   STATUS[774].EXT.BIT19 := FALSE;
   STATUS[774].EXT.BIT20 := FALSE;
   STATUS[774].EXT.AlarmSuppressed := FALSE;
   STATUS[774].EXT.AlarmPrsent := FALSE;
   STATUS[774].EXT.AlarmFailUnAck := FALSE;
   STATUS[774].Status := 0;
   STATUS[774].TimeStamp := 16#0000;
   STATUS[775].VALUE := 0.0;
   STATUS[775].TRIGVALUE := 0.0;
   STATUS[775].EXT.AlarmWarnUnAck := FALSE;
   STATUS[775].EXT.AckRequired := FALSE;
   STATUS[775].EXT.Maintanence := FALSE;
   STATUS[775].EXT.Operation := FALSE;
   STATUS[775].EXT.Forced := FALSE;
   STATUS[775].EXT.BIT29 := FALSE;
   STATUS[775].EXT.BIT30 := FALSE;
   STATUS[775].EXT.BIT31 := FALSE;
   STATUS[775].EXT.ModeBit1 := FALSE;
   STATUS[775].EXT.ModeBit2 := FALSE;
   STATUS[775].EXT.ModeBit3 := FALSE;
   STATUS[775].EXT.BIT19 := FALSE;
   STATUS[775].EXT.BIT20 := FALSE;
   STATUS[775].EXT.AlarmSuppressed := FALSE;
   STATUS[775].EXT.AlarmPrsent := FALSE;
   STATUS[775].EXT.AlarmFailUnAck := FALSE;
   STATUS[775].Status := 0;
   STATUS[775].TimeStamp := 16#0000;
   STATUS[776].VALUE := 0.0;
   STATUS[776].TRIGVALUE := 0.0;
   STATUS[776].EXT.AlarmWarnUnAck := FALSE;
   STATUS[776].EXT.AckRequired := FALSE;
   STATUS[776].EXT.Maintanence := FALSE;
   STATUS[776].EXT.Operation := FALSE;
   STATUS[776].EXT.Forced := FALSE;
   STATUS[776].EXT.BIT29 := FALSE;
   STATUS[776].EXT.BIT30 := FALSE;
   STATUS[776].EXT.BIT31 := FALSE;
   STATUS[776].EXT.ModeBit1 := FALSE;
   STATUS[776].EXT.ModeBit2 := FALSE;
   STATUS[776].EXT.ModeBit3 := FALSE;
   STATUS[776].EXT.BIT19 := FALSE;
   STATUS[776].EXT.BIT20 := FALSE;
   STATUS[776].EXT.AlarmSuppressed := FALSE;
   STATUS[776].EXT.AlarmPrsent := FALSE;
   STATUS[776].EXT.AlarmFailUnAck := FALSE;
   STATUS[776].Status := 0;
   STATUS[776].TimeStamp := 16#0000;
   STATUS[777].VALUE := 0.0;
   STATUS[777].TRIGVALUE := 0.0;
   STATUS[777].EXT.AlarmWarnUnAck := FALSE;
   STATUS[777].EXT.AckRequired := FALSE;
   STATUS[777].EXT.Maintanence := FALSE;
   STATUS[777].EXT.Operation := FALSE;
   STATUS[777].EXT.Forced := FALSE;
   STATUS[777].EXT.BIT29 := FALSE;
   STATUS[777].EXT.BIT30 := FALSE;
   STATUS[777].EXT.BIT31 := FALSE;
   STATUS[777].EXT.ModeBit1 := FALSE;
   STATUS[777].EXT.ModeBit2 := FALSE;
   STATUS[777].EXT.ModeBit3 := FALSE;
   STATUS[777].EXT.BIT19 := FALSE;
   STATUS[777].EXT.BIT20 := FALSE;
   STATUS[777].EXT.AlarmSuppressed := FALSE;
   STATUS[777].EXT.AlarmPrsent := FALSE;
   STATUS[777].EXT.AlarmFailUnAck := FALSE;
   STATUS[777].Status := 0;
   STATUS[777].TimeStamp := 16#0000;
   STATUS[778].VALUE := 0.0;
   STATUS[778].TRIGVALUE := 0.0;
   STATUS[778].EXT.AlarmWarnUnAck := FALSE;
   STATUS[778].EXT.AckRequired := FALSE;
   STATUS[778].EXT.Maintanence := FALSE;
   STATUS[778].EXT.Operation := FALSE;
   STATUS[778].EXT.Forced := FALSE;
   STATUS[778].EXT.BIT29 := FALSE;
   STATUS[778].EXT.BIT30 := FALSE;
   STATUS[778].EXT.BIT31 := FALSE;
   STATUS[778].EXT.ModeBit1 := FALSE;
   STATUS[778].EXT.ModeBit2 := FALSE;
   STATUS[778].EXT.ModeBit3 := FALSE;
   STATUS[778].EXT.BIT19 := FALSE;
   STATUS[778].EXT.BIT20 := FALSE;
   STATUS[778].EXT.AlarmSuppressed := FALSE;
   STATUS[778].EXT.AlarmPrsent := FALSE;
   STATUS[778].EXT.AlarmFailUnAck := FALSE;
   STATUS[778].Status := 0;
   STATUS[778].TimeStamp := 16#0000;
   STATUS[779].VALUE := 0.0;
   STATUS[779].TRIGVALUE := 0.0;
   STATUS[779].EXT.AlarmWarnUnAck := FALSE;
   STATUS[779].EXT.AckRequired := FALSE;
   STATUS[779].EXT.Maintanence := FALSE;
   STATUS[779].EXT.Operation := FALSE;
   STATUS[779].EXT.Forced := FALSE;
   STATUS[779].EXT.BIT29 := FALSE;
   STATUS[779].EXT.BIT30 := FALSE;
   STATUS[779].EXT.BIT31 := FALSE;
   STATUS[779].EXT.ModeBit1 := FALSE;
   STATUS[779].EXT.ModeBit2 := FALSE;
   STATUS[779].EXT.ModeBit3 := FALSE;
   STATUS[779].EXT.BIT19 := FALSE;
   STATUS[779].EXT.BIT20 := FALSE;
   STATUS[779].EXT.AlarmSuppressed := FALSE;
   STATUS[779].EXT.AlarmPrsent := FALSE;
   STATUS[779].EXT.AlarmFailUnAck := FALSE;
   STATUS[779].Status := 0;
   STATUS[779].TimeStamp := 16#0000;
   STATUS[780].VALUE := 0.0;
   STATUS[780].TRIGVALUE := 0.0;
   STATUS[780].EXT.AlarmWarnUnAck := FALSE;
   STATUS[780].EXT.AckRequired := FALSE;
   STATUS[780].EXT.Maintanence := FALSE;
   STATUS[780].EXT.Operation := FALSE;
   STATUS[780].EXT.Forced := FALSE;
   STATUS[780].EXT.BIT29 := FALSE;
   STATUS[780].EXT.BIT30 := FALSE;
   STATUS[780].EXT.BIT31 := FALSE;
   STATUS[780].EXT.ModeBit1 := FALSE;
   STATUS[780].EXT.ModeBit2 := FALSE;
   STATUS[780].EXT.ModeBit3 := FALSE;
   STATUS[780].EXT.BIT19 := FALSE;
   STATUS[780].EXT.BIT20 := FALSE;
   STATUS[780].EXT.AlarmSuppressed := FALSE;
   STATUS[780].EXT.AlarmPrsent := FALSE;
   STATUS[780].EXT.AlarmFailUnAck := FALSE;
   STATUS[780].Status := 0;
   STATUS[780].TimeStamp := 16#0000;
   STATUS[781].VALUE := 0.0;
   STATUS[781].TRIGVALUE := 0.0;
   STATUS[781].EXT.AlarmWarnUnAck := FALSE;
   STATUS[781].EXT.AckRequired := FALSE;
   STATUS[781].EXT.Maintanence := FALSE;
   STATUS[781].EXT.Operation := FALSE;
   STATUS[781].EXT.Forced := FALSE;
   STATUS[781].EXT.BIT29 := FALSE;
   STATUS[781].EXT.BIT30 := FALSE;
   STATUS[781].EXT.BIT31 := FALSE;
   STATUS[781].EXT.ModeBit1 := FALSE;
   STATUS[781].EXT.ModeBit2 := FALSE;
   STATUS[781].EXT.ModeBit3 := FALSE;
   STATUS[781].EXT.BIT19 := FALSE;
   STATUS[781].EXT.BIT20 := FALSE;
   STATUS[781].EXT.AlarmSuppressed := FALSE;
   STATUS[781].EXT.AlarmPrsent := FALSE;
   STATUS[781].EXT.AlarmFailUnAck := FALSE;
   STATUS[781].Status := 0;
   STATUS[781].TimeStamp := 16#0000;
   STATUS[782].VALUE := 0.0;
   STATUS[782].TRIGVALUE := 0.0;
   STATUS[782].EXT.AlarmWarnUnAck := FALSE;
   STATUS[782].EXT.AckRequired := FALSE;
   STATUS[782].EXT.Maintanence := FALSE;
   STATUS[782].EXT.Operation := FALSE;
   STATUS[782].EXT.Forced := FALSE;
   STATUS[782].EXT.BIT29 := FALSE;
   STATUS[782].EXT.BIT30 := FALSE;
   STATUS[782].EXT.BIT31 := FALSE;
   STATUS[782].EXT.ModeBit1 := FALSE;
   STATUS[782].EXT.ModeBit2 := FALSE;
   STATUS[782].EXT.ModeBit3 := FALSE;
   STATUS[782].EXT.BIT19 := FALSE;
   STATUS[782].EXT.BIT20 := FALSE;
   STATUS[782].EXT.AlarmSuppressed := FALSE;
   STATUS[782].EXT.AlarmPrsent := FALSE;
   STATUS[782].EXT.AlarmFailUnAck := FALSE;
   STATUS[782].Status := 0;
   STATUS[782].TimeStamp := 16#0000;
   STATUS[783].VALUE := 0.0;
   STATUS[783].TRIGVALUE := 0.0;
   STATUS[783].EXT.AlarmWarnUnAck := FALSE;
   STATUS[783].EXT.AckRequired := FALSE;
   STATUS[783].EXT.Maintanence := FALSE;
   STATUS[783].EXT.Operation := FALSE;
   STATUS[783].EXT.Forced := FALSE;
   STATUS[783].EXT.BIT29 := FALSE;
   STATUS[783].EXT.BIT30 := FALSE;
   STATUS[783].EXT.BIT31 := FALSE;
   STATUS[783].EXT.ModeBit1 := FALSE;
   STATUS[783].EXT.ModeBit2 := FALSE;
   STATUS[783].EXT.ModeBit3 := FALSE;
   STATUS[783].EXT.BIT19 := FALSE;
   STATUS[783].EXT.BIT20 := FALSE;
   STATUS[783].EXT.AlarmSuppressed := FALSE;
   STATUS[783].EXT.AlarmPrsent := FALSE;
   STATUS[783].EXT.AlarmFailUnAck := FALSE;
   STATUS[783].Status := 0;
   STATUS[783].TimeStamp := 16#0000;
   STATUS[784].VALUE := 0.0;
   STATUS[784].TRIGVALUE := 0.0;
   STATUS[784].EXT.AlarmWarnUnAck := FALSE;
   STATUS[784].EXT.AckRequired := FALSE;
   STATUS[784].EXT.Maintanence := FALSE;
   STATUS[784].EXT.Operation := FALSE;
   STATUS[784].EXT.Forced := FALSE;
   STATUS[784].EXT.BIT29 := FALSE;
   STATUS[784].EXT.BIT30 := FALSE;
   STATUS[784].EXT.BIT31 := FALSE;
   STATUS[784].EXT.ModeBit1 := FALSE;
   STATUS[784].EXT.ModeBit2 := FALSE;
   STATUS[784].EXT.ModeBit3 := FALSE;
   STATUS[784].EXT.BIT19 := FALSE;
   STATUS[784].EXT.BIT20 := FALSE;
   STATUS[784].EXT.AlarmSuppressed := FALSE;
   STATUS[784].EXT.AlarmPrsent := FALSE;
   STATUS[784].EXT.AlarmFailUnAck := FALSE;
   STATUS[784].Status := 0;
   STATUS[784].TimeStamp := 16#0000;
   STATUS[785].VALUE := 0.0;
   STATUS[785].TRIGVALUE := 0.0;
   STATUS[785].EXT.AlarmWarnUnAck := FALSE;
   STATUS[785].EXT.AckRequired := FALSE;
   STATUS[785].EXT.Maintanence := FALSE;
   STATUS[785].EXT.Operation := FALSE;
   STATUS[785].EXT.Forced := FALSE;
   STATUS[785].EXT.BIT29 := FALSE;
   STATUS[785].EXT.BIT30 := FALSE;
   STATUS[785].EXT.BIT31 := FALSE;
   STATUS[785].EXT.ModeBit1 := FALSE;
   STATUS[785].EXT.ModeBit2 := FALSE;
   STATUS[785].EXT.ModeBit3 := FALSE;
   STATUS[785].EXT.BIT19 := FALSE;
   STATUS[785].EXT.BIT20 := FALSE;
   STATUS[785].EXT.AlarmSuppressed := FALSE;
   STATUS[785].EXT.AlarmPrsent := FALSE;
   STATUS[785].EXT.AlarmFailUnAck := FALSE;
   STATUS[785].Status := 0;
   STATUS[785].TimeStamp := 16#0000;
   STATUS[786].VALUE := 0.0;
   STATUS[786].TRIGVALUE := 0.0;
   STATUS[786].EXT.AlarmWarnUnAck := FALSE;
   STATUS[786].EXT.AckRequired := FALSE;
   STATUS[786].EXT.Maintanence := FALSE;
   STATUS[786].EXT.Operation := FALSE;
   STATUS[786].EXT.Forced := FALSE;
   STATUS[786].EXT.BIT29 := FALSE;
   STATUS[786].EXT.BIT30 := FALSE;
   STATUS[786].EXT.BIT31 := FALSE;
   STATUS[786].EXT.ModeBit1 := FALSE;
   STATUS[786].EXT.ModeBit2 := FALSE;
   STATUS[786].EXT.ModeBit3 := FALSE;
   STATUS[786].EXT.BIT19 := FALSE;
   STATUS[786].EXT.BIT20 := FALSE;
   STATUS[786].EXT.AlarmSuppressed := FALSE;
   STATUS[786].EXT.AlarmPrsent := FALSE;
   STATUS[786].EXT.AlarmFailUnAck := FALSE;
   STATUS[786].Status := 0;
   STATUS[786].TimeStamp := 16#0000;
   STATUS[787].VALUE := 0.0;
   STATUS[787].TRIGVALUE := 0.0;
   STATUS[787].EXT.AlarmWarnUnAck := FALSE;
   STATUS[787].EXT.AckRequired := FALSE;
   STATUS[787].EXT.Maintanence := FALSE;
   STATUS[787].EXT.Operation := FALSE;
   STATUS[787].EXT.Forced := FALSE;
   STATUS[787].EXT.BIT29 := FALSE;
   STATUS[787].EXT.BIT30 := FALSE;
   STATUS[787].EXT.BIT31 := FALSE;
   STATUS[787].EXT.ModeBit1 := FALSE;
   STATUS[787].EXT.ModeBit2 := FALSE;
   STATUS[787].EXT.ModeBit3 := FALSE;
   STATUS[787].EXT.BIT19 := FALSE;
   STATUS[787].EXT.BIT20 := FALSE;
   STATUS[787].EXT.AlarmSuppressed := FALSE;
   STATUS[787].EXT.AlarmPrsent := FALSE;
   STATUS[787].EXT.AlarmFailUnAck := FALSE;
   STATUS[787].Status := 0;
   STATUS[787].TimeStamp := 16#0000;
   STATUS[788].VALUE := 0.0;
   STATUS[788].TRIGVALUE := 0.0;
   STATUS[788].EXT.AlarmWarnUnAck := FALSE;
   STATUS[788].EXT.AckRequired := FALSE;
   STATUS[788].EXT.Maintanence := FALSE;
   STATUS[788].EXT.Operation := FALSE;
   STATUS[788].EXT.Forced := FALSE;
   STATUS[788].EXT.BIT29 := FALSE;
   STATUS[788].EXT.BIT30 := FALSE;
   STATUS[788].EXT.BIT31 := FALSE;
   STATUS[788].EXT.ModeBit1 := FALSE;
   STATUS[788].EXT.ModeBit2 := FALSE;
   STATUS[788].EXT.ModeBit3 := FALSE;
   STATUS[788].EXT.BIT19 := FALSE;
   STATUS[788].EXT.BIT20 := FALSE;
   STATUS[788].EXT.AlarmSuppressed := FALSE;
   STATUS[788].EXT.AlarmPrsent := FALSE;
   STATUS[788].EXT.AlarmFailUnAck := FALSE;
   STATUS[788].Status := 0;
   STATUS[788].TimeStamp := 16#0000;
   STATUS[789].VALUE := 0.0;
   STATUS[789].TRIGVALUE := 0.0;
   STATUS[789].EXT.AlarmWarnUnAck := FALSE;
   STATUS[789].EXT.AckRequired := FALSE;
   STATUS[789].EXT.Maintanence := FALSE;
   STATUS[789].EXT.Operation := FALSE;
   STATUS[789].EXT.Forced := FALSE;
   STATUS[789].EXT.BIT29 := FALSE;
   STATUS[789].EXT.BIT30 := FALSE;
   STATUS[789].EXT.BIT31 := FALSE;
   STATUS[789].EXT.ModeBit1 := FALSE;
   STATUS[789].EXT.ModeBit2 := FALSE;
   STATUS[789].EXT.ModeBit3 := FALSE;
   STATUS[789].EXT.BIT19 := FALSE;
   STATUS[789].EXT.BIT20 := FALSE;
   STATUS[789].EXT.AlarmSuppressed := FALSE;
   STATUS[789].EXT.AlarmPrsent := FALSE;
   STATUS[789].EXT.AlarmFailUnAck := FALSE;
   STATUS[789].Status := 0;
   STATUS[789].TimeStamp := 16#0000;
   STATUS[790].VALUE := 0.0;
   STATUS[790].TRIGVALUE := 0.0;
   STATUS[790].EXT.AlarmWarnUnAck := FALSE;
   STATUS[790].EXT.AckRequired := FALSE;
   STATUS[790].EXT.Maintanence := FALSE;
   STATUS[790].EXT.Operation := FALSE;
   STATUS[790].EXT.Forced := FALSE;
   STATUS[790].EXT.BIT29 := FALSE;
   STATUS[790].EXT.BIT30 := FALSE;
   STATUS[790].EXT.BIT31 := FALSE;
   STATUS[790].EXT.ModeBit1 := FALSE;
   STATUS[790].EXT.ModeBit2 := FALSE;
   STATUS[790].EXT.ModeBit3 := FALSE;
   STATUS[790].EXT.BIT19 := FALSE;
   STATUS[790].EXT.BIT20 := FALSE;
   STATUS[790].EXT.AlarmSuppressed := FALSE;
   STATUS[790].EXT.AlarmPrsent := FALSE;
   STATUS[790].EXT.AlarmFailUnAck := FALSE;
   STATUS[790].Status := 0;
   STATUS[790].TimeStamp := 16#0000;
   STATUS[791].VALUE := 0.0;
   STATUS[791].TRIGVALUE := 0.0;
   STATUS[791].EXT.AlarmWarnUnAck := FALSE;
   STATUS[791].EXT.AckRequired := FALSE;
   STATUS[791].EXT.Maintanence := FALSE;
   STATUS[791].EXT.Operation := FALSE;
   STATUS[791].EXT.Forced := FALSE;
   STATUS[791].EXT.BIT29 := FALSE;
   STATUS[791].EXT.BIT30 := FALSE;
   STATUS[791].EXT.BIT31 := FALSE;
   STATUS[791].EXT.ModeBit1 := FALSE;
   STATUS[791].EXT.ModeBit2 := FALSE;
   STATUS[791].EXT.ModeBit3 := FALSE;
   STATUS[791].EXT.BIT19 := FALSE;
   STATUS[791].EXT.BIT20 := FALSE;
   STATUS[791].EXT.AlarmSuppressed := FALSE;
   STATUS[791].EXT.AlarmPrsent := FALSE;
   STATUS[791].EXT.AlarmFailUnAck := FALSE;
   STATUS[791].Status := 0;
   STATUS[791].TimeStamp := 16#0000;
   STATUS[792].VALUE := 0.0;
   STATUS[792].TRIGVALUE := 0.0;
   STATUS[792].EXT.AlarmWarnUnAck := FALSE;
   STATUS[792].EXT.AckRequired := FALSE;
   STATUS[792].EXT.Maintanence := FALSE;
   STATUS[792].EXT.Operation := FALSE;
   STATUS[792].EXT.Forced := FALSE;
   STATUS[792].EXT.BIT29 := FALSE;
   STATUS[792].EXT.BIT30 := FALSE;
   STATUS[792].EXT.BIT31 := FALSE;
   STATUS[792].EXT.ModeBit1 := FALSE;
   STATUS[792].EXT.ModeBit2 := FALSE;
   STATUS[792].EXT.ModeBit3 := FALSE;
   STATUS[792].EXT.BIT19 := FALSE;
   STATUS[792].EXT.BIT20 := FALSE;
   STATUS[792].EXT.AlarmSuppressed := FALSE;
   STATUS[792].EXT.AlarmPrsent := FALSE;
   STATUS[792].EXT.AlarmFailUnAck := FALSE;
   STATUS[792].Status := 0;
   STATUS[792].TimeStamp := 16#0000;
   STATUS[793].VALUE := 0.0;
   STATUS[793].TRIGVALUE := 0.0;
   STATUS[793].EXT.AlarmWarnUnAck := FALSE;
   STATUS[793].EXT.AckRequired := FALSE;
   STATUS[793].EXT.Maintanence := FALSE;
   STATUS[793].EXT.Operation := FALSE;
   STATUS[793].EXT.Forced := FALSE;
   STATUS[793].EXT.BIT29 := FALSE;
   STATUS[793].EXT.BIT30 := FALSE;
   STATUS[793].EXT.BIT31 := FALSE;
   STATUS[793].EXT.ModeBit1 := FALSE;
   STATUS[793].EXT.ModeBit2 := FALSE;
   STATUS[793].EXT.ModeBit3 := FALSE;
   STATUS[793].EXT.BIT19 := FALSE;
   STATUS[793].EXT.BIT20 := FALSE;
   STATUS[793].EXT.AlarmSuppressed := FALSE;
   STATUS[793].EXT.AlarmPrsent := FALSE;
   STATUS[793].EXT.AlarmFailUnAck := FALSE;
   STATUS[793].Status := 0;
   STATUS[793].TimeStamp := 16#0000;
   STATUS[794].VALUE := 0.0;
   STATUS[794].TRIGVALUE := 0.0;
   STATUS[794].EXT.AlarmWarnUnAck := FALSE;
   STATUS[794].EXT.AckRequired := FALSE;
   STATUS[794].EXT.Maintanence := FALSE;
   STATUS[794].EXT.Operation := FALSE;
   STATUS[794].EXT.Forced := FALSE;
   STATUS[794].EXT.BIT29 := FALSE;
   STATUS[794].EXT.BIT30 := FALSE;
   STATUS[794].EXT.BIT31 := FALSE;
   STATUS[794].EXT.ModeBit1 := FALSE;
   STATUS[794].EXT.ModeBit2 := FALSE;
   STATUS[794].EXT.ModeBit3 := FALSE;
   STATUS[794].EXT.BIT19 := FALSE;
   STATUS[794].EXT.BIT20 := FALSE;
   STATUS[794].EXT.AlarmSuppressed := FALSE;
   STATUS[794].EXT.AlarmPrsent := FALSE;
   STATUS[794].EXT.AlarmFailUnAck := FALSE;
   STATUS[794].Status := 0;
   STATUS[794].TimeStamp := 16#0000;
   STATUS[795].VALUE := 0.0;
   STATUS[795].TRIGVALUE := 0.0;
   STATUS[795].EXT.AlarmWarnUnAck := FALSE;
   STATUS[795].EXT.AckRequired := FALSE;
   STATUS[795].EXT.Maintanence := FALSE;
   STATUS[795].EXT.Operation := FALSE;
   STATUS[795].EXT.Forced := FALSE;
   STATUS[795].EXT.BIT29 := FALSE;
   STATUS[795].EXT.BIT30 := FALSE;
   STATUS[795].EXT.BIT31 := FALSE;
   STATUS[795].EXT.ModeBit1 := FALSE;
   STATUS[795].EXT.ModeBit2 := FALSE;
   STATUS[795].EXT.ModeBit3 := FALSE;
   STATUS[795].EXT.BIT19 := FALSE;
   STATUS[795].EXT.BIT20 := FALSE;
   STATUS[795].EXT.AlarmSuppressed := FALSE;
   STATUS[795].EXT.AlarmPrsent := FALSE;
   STATUS[795].EXT.AlarmFailUnAck := FALSE;
   STATUS[795].Status := 0;
   STATUS[795].TimeStamp := 16#0000;
   STATUS[796].VALUE := 0.0;
   STATUS[796].TRIGVALUE := 0.0;
   STATUS[796].EXT.AlarmWarnUnAck := FALSE;
   STATUS[796].EXT.AckRequired := FALSE;
   STATUS[796].EXT.Maintanence := FALSE;
   STATUS[796].EXT.Operation := FALSE;
   STATUS[796].EXT.Forced := FALSE;
   STATUS[796].EXT.BIT29 := FALSE;
   STATUS[796].EXT.BIT30 := FALSE;
   STATUS[796].EXT.BIT31 := FALSE;
   STATUS[796].EXT.ModeBit1 := FALSE;
   STATUS[796].EXT.ModeBit2 := FALSE;
   STATUS[796].EXT.ModeBit3 := FALSE;
   STATUS[796].EXT.BIT19 := FALSE;
   STATUS[796].EXT.BIT20 := FALSE;
   STATUS[796].EXT.AlarmSuppressed := FALSE;
   STATUS[796].EXT.AlarmPrsent := FALSE;
   STATUS[796].EXT.AlarmFailUnAck := FALSE;
   STATUS[796].Status := 0;
   STATUS[796].TimeStamp := 16#0000;
   STATUS[797].VALUE := 0.0;
   STATUS[797].TRIGVALUE := 0.0;
   STATUS[797].EXT.AlarmWarnUnAck := FALSE;
   STATUS[797].EXT.AckRequired := FALSE;
   STATUS[797].EXT.Maintanence := FALSE;
   STATUS[797].EXT.Operation := FALSE;
   STATUS[797].EXT.Forced := FALSE;
   STATUS[797].EXT.BIT29 := FALSE;
   STATUS[797].EXT.BIT30 := FALSE;
   STATUS[797].EXT.BIT31 := FALSE;
   STATUS[797].EXT.ModeBit1 := FALSE;
   STATUS[797].EXT.ModeBit2 := FALSE;
   STATUS[797].EXT.ModeBit3 := FALSE;
   STATUS[797].EXT.BIT19 := FALSE;
   STATUS[797].EXT.BIT20 := FALSE;
   STATUS[797].EXT.AlarmSuppressed := FALSE;
   STATUS[797].EXT.AlarmPrsent := FALSE;
   STATUS[797].EXT.AlarmFailUnAck := FALSE;
   STATUS[797].Status := 0;
   STATUS[797].TimeStamp := 16#0000;
   STATUS[798].VALUE := 0.0;
   STATUS[798].TRIGVALUE := 0.0;
   STATUS[798].EXT.AlarmWarnUnAck := FALSE;
   STATUS[798].EXT.AckRequired := FALSE;
   STATUS[798].EXT.Maintanence := FALSE;
   STATUS[798].EXT.Operation := FALSE;
   STATUS[798].EXT.Forced := FALSE;
   STATUS[798].EXT.BIT29 := FALSE;
   STATUS[798].EXT.BIT30 := FALSE;
   STATUS[798].EXT.BIT31 := FALSE;
   STATUS[798].EXT.ModeBit1 := FALSE;
   STATUS[798].EXT.ModeBit2 := FALSE;
   STATUS[798].EXT.ModeBit3 := FALSE;
   STATUS[798].EXT.BIT19 := FALSE;
   STATUS[798].EXT.BIT20 := FALSE;
   STATUS[798].EXT.AlarmSuppressed := FALSE;
   STATUS[798].EXT.AlarmPrsent := FALSE;
   STATUS[798].EXT.AlarmFailUnAck := FALSE;
   STATUS[798].Status := 0;
   STATUS[798].TimeStamp := 16#0000;
   STATUS[799].VALUE := 0.0;
   STATUS[799].TRIGVALUE := 0.0;
   STATUS[799].EXT.AlarmWarnUnAck := FALSE;
   STATUS[799].EXT.AckRequired := FALSE;
   STATUS[799].EXT.Maintanence := FALSE;
   STATUS[799].EXT.Operation := FALSE;
   STATUS[799].EXT.Forced := FALSE;
   STATUS[799].EXT.BIT29 := FALSE;
   STATUS[799].EXT.BIT30 := FALSE;
   STATUS[799].EXT.BIT31 := FALSE;
   STATUS[799].EXT.ModeBit1 := FALSE;
   STATUS[799].EXT.ModeBit2 := FALSE;
   STATUS[799].EXT.ModeBit3 := FALSE;
   STATUS[799].EXT.BIT19 := FALSE;
   STATUS[799].EXT.BIT20 := FALSE;
   STATUS[799].EXT.AlarmSuppressed := FALSE;
   STATUS[799].EXT.AlarmPrsent := FALSE;
   STATUS[799].EXT.AlarmFailUnAck := FALSE;
   STATUS[799].Status := 0;
   STATUS[799].TimeStamp := 16#0000;
   STATUS[800].VALUE := 0.0;
   STATUS[800].TRIGVALUE := 0.0;
   STATUS[800].EXT.AlarmWarnUnAck := FALSE;
   STATUS[800].EXT.AckRequired := FALSE;
   STATUS[800].EXT.Maintanence := FALSE;
   STATUS[800].EXT.Operation := FALSE;
   STATUS[800].EXT.Forced := FALSE;
   STATUS[800].EXT.BIT29 := FALSE;
   STATUS[800].EXT.BIT30 := FALSE;
   STATUS[800].EXT.BIT31 := FALSE;
   STATUS[800].EXT.ModeBit1 := FALSE;
   STATUS[800].EXT.ModeBit2 := FALSE;
   STATUS[800].EXT.ModeBit3 := FALSE;
   STATUS[800].EXT.BIT19 := FALSE;
   STATUS[800].EXT.BIT20 := FALSE;
   STATUS[800].EXT.AlarmSuppressed := FALSE;
   STATUS[800].EXT.AlarmPrsent := FALSE;
   STATUS[800].EXT.AlarmFailUnAck := FALSE;
   STATUS[800].Status := 0;
   STATUS[800].TimeStamp := 16#0000;
   STATUS[801].VALUE := 0.0;
   STATUS[801].TRIGVALUE := 0.0;
   STATUS[801].EXT.AlarmWarnUnAck := FALSE;
   STATUS[801].EXT.AckRequired := FALSE;
   STATUS[801].EXT.Maintanence := FALSE;
   STATUS[801].EXT.Operation := FALSE;
   STATUS[801].EXT.Forced := FALSE;
   STATUS[801].EXT.BIT29 := FALSE;
   STATUS[801].EXT.BIT30 := FALSE;
   STATUS[801].EXT.BIT31 := FALSE;
   STATUS[801].EXT.ModeBit1 := FALSE;
   STATUS[801].EXT.ModeBit2 := FALSE;
   STATUS[801].EXT.ModeBit3 := FALSE;
   STATUS[801].EXT.BIT19 := FALSE;
   STATUS[801].EXT.BIT20 := FALSE;
   STATUS[801].EXT.AlarmSuppressed := FALSE;
   STATUS[801].EXT.AlarmPrsent := FALSE;
   STATUS[801].EXT.AlarmFailUnAck := FALSE;
   STATUS[801].Status := 0;
   STATUS[801].TimeStamp := 16#0000;
   STATUS[802].VALUE := 0.0;
   STATUS[802].TRIGVALUE := 0.0;
   STATUS[802].EXT.AlarmWarnUnAck := FALSE;
   STATUS[802].EXT.AckRequired := FALSE;
   STATUS[802].EXT.Maintanence := FALSE;
   STATUS[802].EXT.Operation := FALSE;
   STATUS[802].EXT.Forced := FALSE;
   STATUS[802].EXT.BIT29 := FALSE;
   STATUS[802].EXT.BIT30 := FALSE;
   STATUS[802].EXT.BIT31 := FALSE;
   STATUS[802].EXT.ModeBit1 := FALSE;
   STATUS[802].EXT.ModeBit2 := FALSE;
   STATUS[802].EXT.ModeBit3 := FALSE;
   STATUS[802].EXT.BIT19 := FALSE;
   STATUS[802].EXT.BIT20 := FALSE;
   STATUS[802].EXT.AlarmSuppressed := FALSE;
   STATUS[802].EXT.AlarmPrsent := FALSE;
   STATUS[802].EXT.AlarmFailUnAck := FALSE;
   STATUS[802].Status := 0;
   STATUS[802].TimeStamp := 16#0000;
   STATUS[803].VALUE := 0.0;
   STATUS[803].TRIGVALUE := 0.0;
   STATUS[803].EXT.AlarmWarnUnAck := FALSE;
   STATUS[803].EXT.AckRequired := FALSE;
   STATUS[803].EXT.Maintanence := FALSE;
   STATUS[803].EXT.Operation := FALSE;
   STATUS[803].EXT.Forced := FALSE;
   STATUS[803].EXT.BIT29 := FALSE;
   STATUS[803].EXT.BIT30 := FALSE;
   STATUS[803].EXT.BIT31 := FALSE;
   STATUS[803].EXT.ModeBit1 := FALSE;
   STATUS[803].EXT.ModeBit2 := FALSE;
   STATUS[803].EXT.ModeBit3 := FALSE;
   STATUS[803].EXT.BIT19 := FALSE;
   STATUS[803].EXT.BIT20 := FALSE;
   STATUS[803].EXT.AlarmSuppressed := FALSE;
   STATUS[803].EXT.AlarmPrsent := FALSE;
   STATUS[803].EXT.AlarmFailUnAck := FALSE;
   STATUS[803].Status := 0;
   STATUS[803].TimeStamp := 16#0000;
   STATUS[804].VALUE := 0.0;
   STATUS[804].TRIGVALUE := 0.0;
   STATUS[804].EXT.AlarmWarnUnAck := FALSE;
   STATUS[804].EXT.AckRequired := FALSE;
   STATUS[804].EXT.Maintanence := FALSE;
   STATUS[804].EXT.Operation := FALSE;
   STATUS[804].EXT.Forced := FALSE;
   STATUS[804].EXT.BIT29 := FALSE;
   STATUS[804].EXT.BIT30 := FALSE;
   STATUS[804].EXT.BIT31 := FALSE;
   STATUS[804].EXT.ModeBit1 := FALSE;
   STATUS[804].EXT.ModeBit2 := FALSE;
   STATUS[804].EXT.ModeBit3 := FALSE;
   STATUS[804].EXT.BIT19 := FALSE;
   STATUS[804].EXT.BIT20 := FALSE;
   STATUS[804].EXT.AlarmSuppressed := FALSE;
   STATUS[804].EXT.AlarmPrsent := FALSE;
   STATUS[804].EXT.AlarmFailUnAck := FALSE;
   STATUS[804].Status := 0;
   STATUS[804].TimeStamp := 16#0000;
   STATUS[805].VALUE := 0.0;
   STATUS[805].TRIGVALUE := 0.0;
   STATUS[805].EXT.AlarmWarnUnAck := FALSE;
   STATUS[805].EXT.AckRequired := FALSE;
   STATUS[805].EXT.Maintanence := FALSE;
   STATUS[805].EXT.Operation := FALSE;
   STATUS[805].EXT.Forced := FALSE;
   STATUS[805].EXT.BIT29 := FALSE;
   STATUS[805].EXT.BIT30 := FALSE;
   STATUS[805].EXT.BIT31 := FALSE;
   STATUS[805].EXT.ModeBit1 := FALSE;
   STATUS[805].EXT.ModeBit2 := FALSE;
   STATUS[805].EXT.ModeBit3 := FALSE;
   STATUS[805].EXT.BIT19 := FALSE;
   STATUS[805].EXT.BIT20 := FALSE;
   STATUS[805].EXT.AlarmSuppressed := FALSE;
   STATUS[805].EXT.AlarmPrsent := FALSE;
   STATUS[805].EXT.AlarmFailUnAck := FALSE;
   STATUS[805].Status := 0;
   STATUS[805].TimeStamp := 16#0000;
   STATUS[806].VALUE := 0.0;
   STATUS[806].TRIGVALUE := 0.0;
   STATUS[806].EXT.AlarmWarnUnAck := FALSE;
   STATUS[806].EXT.AckRequired := FALSE;
   STATUS[806].EXT.Maintanence := FALSE;
   STATUS[806].EXT.Operation := FALSE;
   STATUS[806].EXT.Forced := FALSE;
   STATUS[806].EXT.BIT29 := FALSE;
   STATUS[806].EXT.BIT30 := FALSE;
   STATUS[806].EXT.BIT31 := FALSE;
   STATUS[806].EXT.ModeBit1 := FALSE;
   STATUS[806].EXT.ModeBit2 := FALSE;
   STATUS[806].EXT.ModeBit3 := FALSE;
   STATUS[806].EXT.BIT19 := FALSE;
   STATUS[806].EXT.BIT20 := FALSE;
   STATUS[806].EXT.AlarmSuppressed := FALSE;
   STATUS[806].EXT.AlarmPrsent := FALSE;
   STATUS[806].EXT.AlarmFailUnAck := FALSE;
   STATUS[806].Status := 0;
   STATUS[806].TimeStamp := 16#0000;
   STATUS[807].VALUE := 0.0;
   STATUS[807].TRIGVALUE := 0.0;
   STATUS[807].EXT.AlarmWarnUnAck := FALSE;
   STATUS[807].EXT.AckRequired := FALSE;
   STATUS[807].EXT.Maintanence := FALSE;
   STATUS[807].EXT.Operation := FALSE;
   STATUS[807].EXT.Forced := FALSE;
   STATUS[807].EXT.BIT29 := FALSE;
   STATUS[807].EXT.BIT30 := FALSE;
   STATUS[807].EXT.BIT31 := FALSE;
   STATUS[807].EXT.ModeBit1 := FALSE;
   STATUS[807].EXT.ModeBit2 := FALSE;
   STATUS[807].EXT.ModeBit3 := FALSE;
   STATUS[807].EXT.BIT19 := FALSE;
   STATUS[807].EXT.BIT20 := FALSE;
   STATUS[807].EXT.AlarmSuppressed := FALSE;
   STATUS[807].EXT.AlarmPrsent := FALSE;
   STATUS[807].EXT.AlarmFailUnAck := FALSE;
   STATUS[807].Status := 0;
   STATUS[807].TimeStamp := 16#0000;
   STATUS[808].VALUE := 0.0;
   STATUS[808].TRIGVALUE := 0.0;
   STATUS[808].EXT.AlarmWarnUnAck := FALSE;
   STATUS[808].EXT.AckRequired := FALSE;
   STATUS[808].EXT.Maintanence := FALSE;
   STATUS[808].EXT.Operation := FALSE;
   STATUS[808].EXT.Forced := FALSE;
   STATUS[808].EXT.BIT29 := FALSE;
   STATUS[808].EXT.BIT30 := FALSE;
   STATUS[808].EXT.BIT31 := FALSE;
   STATUS[808].EXT.ModeBit1 := FALSE;
   STATUS[808].EXT.ModeBit2 := FALSE;
   STATUS[808].EXT.ModeBit3 := FALSE;
   STATUS[808].EXT.BIT19 := FALSE;
   STATUS[808].EXT.BIT20 := FALSE;
   STATUS[808].EXT.AlarmSuppressed := FALSE;
   STATUS[808].EXT.AlarmPrsent := FALSE;
   STATUS[808].EXT.AlarmFailUnAck := FALSE;
   STATUS[808].Status := 0;
   STATUS[808].TimeStamp := 16#0000;
   STATUS[809].VALUE := 0.0;
   STATUS[809].TRIGVALUE := 0.0;
   STATUS[809].EXT.AlarmWarnUnAck := FALSE;
   STATUS[809].EXT.AckRequired := FALSE;
   STATUS[809].EXT.Maintanence := FALSE;
   STATUS[809].EXT.Operation := FALSE;
   STATUS[809].EXT.Forced := FALSE;
   STATUS[809].EXT.BIT29 := FALSE;
   STATUS[809].EXT.BIT30 := FALSE;
   STATUS[809].EXT.BIT31 := FALSE;
   STATUS[809].EXT.ModeBit1 := FALSE;
   STATUS[809].EXT.ModeBit2 := FALSE;
   STATUS[809].EXT.ModeBit3 := FALSE;
   STATUS[809].EXT.BIT19 := FALSE;
   STATUS[809].EXT.BIT20 := FALSE;
   STATUS[809].EXT.AlarmSuppressed := FALSE;
   STATUS[809].EXT.AlarmPrsent := FALSE;
   STATUS[809].EXT.AlarmFailUnAck := FALSE;
   STATUS[809].Status := 0;
   STATUS[809].TimeStamp := 16#0000;
   STATUS[810].VALUE := 0.0;
   STATUS[810].TRIGVALUE := 0.0;
   STATUS[810].EXT.AlarmWarnUnAck := FALSE;
   STATUS[810].EXT.AckRequired := FALSE;
   STATUS[810].EXT.Maintanence := FALSE;
   STATUS[810].EXT.Operation := FALSE;
   STATUS[810].EXT.Forced := FALSE;
   STATUS[810].EXT.BIT29 := FALSE;
   STATUS[810].EXT.BIT30 := FALSE;
   STATUS[810].EXT.BIT31 := FALSE;
   STATUS[810].EXT.ModeBit1 := FALSE;
   STATUS[810].EXT.ModeBit2 := FALSE;
   STATUS[810].EXT.ModeBit3 := FALSE;
   STATUS[810].EXT.BIT19 := FALSE;
   STATUS[810].EXT.BIT20 := FALSE;
   STATUS[810].EXT.AlarmSuppressed := FALSE;
   STATUS[810].EXT.AlarmPrsent := FALSE;
   STATUS[810].EXT.AlarmFailUnAck := FALSE;
   STATUS[810].Status := 0;
   STATUS[810].TimeStamp := 16#0000;
   STATUS[811].VALUE := 0.0;
   STATUS[811].TRIGVALUE := 0.0;
   STATUS[811].EXT.AlarmWarnUnAck := FALSE;
   STATUS[811].EXT.AckRequired := FALSE;
   STATUS[811].EXT.Maintanence := FALSE;
   STATUS[811].EXT.Operation := FALSE;
   STATUS[811].EXT.Forced := FALSE;
   STATUS[811].EXT.BIT29 := FALSE;
   STATUS[811].EXT.BIT30 := FALSE;
   STATUS[811].EXT.BIT31 := FALSE;
   STATUS[811].EXT.ModeBit1 := FALSE;
   STATUS[811].EXT.ModeBit2 := FALSE;
   STATUS[811].EXT.ModeBit3 := FALSE;
   STATUS[811].EXT.BIT19 := FALSE;
   STATUS[811].EXT.BIT20 := FALSE;
   STATUS[811].EXT.AlarmSuppressed := FALSE;
   STATUS[811].EXT.AlarmPrsent := FALSE;
   STATUS[811].EXT.AlarmFailUnAck := FALSE;
   STATUS[811].Status := 0;
   STATUS[811].TimeStamp := 16#0000;
   STATUS[812].VALUE := 0.0;
   STATUS[812].TRIGVALUE := 0.0;
   STATUS[812].EXT.AlarmWarnUnAck := FALSE;
   STATUS[812].EXT.AckRequired := FALSE;
   STATUS[812].EXT.Maintanence := FALSE;
   STATUS[812].EXT.Operation := FALSE;
   STATUS[812].EXT.Forced := FALSE;
   STATUS[812].EXT.BIT29 := FALSE;
   STATUS[812].EXT.BIT30 := FALSE;
   STATUS[812].EXT.BIT31 := FALSE;
   STATUS[812].EXT.ModeBit1 := FALSE;
   STATUS[812].EXT.ModeBit2 := FALSE;
   STATUS[812].EXT.ModeBit3 := FALSE;
   STATUS[812].EXT.BIT19 := FALSE;
   STATUS[812].EXT.BIT20 := FALSE;
   STATUS[812].EXT.AlarmSuppressed := FALSE;
   STATUS[812].EXT.AlarmPrsent := FALSE;
   STATUS[812].EXT.AlarmFailUnAck := FALSE;
   STATUS[812].Status := 0;
   STATUS[812].TimeStamp := 16#0000;
   STATUS[813].VALUE := 0.0;
   STATUS[813].TRIGVALUE := 0.0;
   STATUS[813].EXT.AlarmWarnUnAck := FALSE;
   STATUS[813].EXT.AckRequired := FALSE;
   STATUS[813].EXT.Maintanence := FALSE;
   STATUS[813].EXT.Operation := FALSE;
   STATUS[813].EXT.Forced := FALSE;
   STATUS[813].EXT.BIT29 := FALSE;
   STATUS[813].EXT.BIT30 := FALSE;
   STATUS[813].EXT.BIT31 := FALSE;
   STATUS[813].EXT.ModeBit1 := FALSE;
   STATUS[813].EXT.ModeBit2 := FALSE;
   STATUS[813].EXT.ModeBit3 := FALSE;
   STATUS[813].EXT.BIT19 := FALSE;
   STATUS[813].EXT.BIT20 := FALSE;
   STATUS[813].EXT.AlarmSuppressed := FALSE;
   STATUS[813].EXT.AlarmPrsent := FALSE;
   STATUS[813].EXT.AlarmFailUnAck := FALSE;
   STATUS[813].Status := 0;
   STATUS[813].TimeStamp := 16#0000;
   STATUS[814].VALUE := 0.0;
   STATUS[814].TRIGVALUE := 0.0;
   STATUS[814].EXT.AlarmWarnUnAck := FALSE;
   STATUS[814].EXT.AckRequired := FALSE;
   STATUS[814].EXT.Maintanence := FALSE;
   STATUS[814].EXT.Operation := FALSE;
   STATUS[814].EXT.Forced := FALSE;
   STATUS[814].EXT.BIT29 := FALSE;
   STATUS[814].EXT.BIT30 := FALSE;
   STATUS[814].EXT.BIT31 := FALSE;
   STATUS[814].EXT.ModeBit1 := FALSE;
   STATUS[814].EXT.ModeBit2 := FALSE;
   STATUS[814].EXT.ModeBit3 := FALSE;
   STATUS[814].EXT.BIT19 := FALSE;
   STATUS[814].EXT.BIT20 := FALSE;
   STATUS[814].EXT.AlarmSuppressed := FALSE;
   STATUS[814].EXT.AlarmPrsent := FALSE;
   STATUS[814].EXT.AlarmFailUnAck := FALSE;
   STATUS[814].Status := 0;
   STATUS[814].TimeStamp := 16#0000;
   STATUS[815].VALUE := 0.0;
   STATUS[815].TRIGVALUE := 0.0;
   STATUS[815].EXT.AlarmWarnUnAck := FALSE;
   STATUS[815].EXT.AckRequired := FALSE;
   STATUS[815].EXT.Maintanence := FALSE;
   STATUS[815].EXT.Operation := FALSE;
   STATUS[815].EXT.Forced := FALSE;
   STATUS[815].EXT.BIT29 := FALSE;
   STATUS[815].EXT.BIT30 := FALSE;
   STATUS[815].EXT.BIT31 := FALSE;
   STATUS[815].EXT.ModeBit1 := FALSE;
   STATUS[815].EXT.ModeBit2 := FALSE;
   STATUS[815].EXT.ModeBit3 := FALSE;
   STATUS[815].EXT.BIT19 := FALSE;
   STATUS[815].EXT.BIT20 := FALSE;
   STATUS[815].EXT.AlarmSuppressed := FALSE;
   STATUS[815].EXT.AlarmPrsent := FALSE;
   STATUS[815].EXT.AlarmFailUnAck := FALSE;
   STATUS[815].Status := 0;
   STATUS[815].TimeStamp := 16#0000;
   STATUS[816].VALUE := 0.0;
   STATUS[816].TRIGVALUE := 0.0;
   STATUS[816].EXT.AlarmWarnUnAck := FALSE;
   STATUS[816].EXT.AckRequired := FALSE;
   STATUS[816].EXT.Maintanence := FALSE;
   STATUS[816].EXT.Operation := FALSE;
   STATUS[816].EXT.Forced := FALSE;
   STATUS[816].EXT.BIT29 := FALSE;
   STATUS[816].EXT.BIT30 := FALSE;
   STATUS[816].EXT.BIT31 := FALSE;
   STATUS[816].EXT.ModeBit1 := FALSE;
   STATUS[816].EXT.ModeBit2 := FALSE;
   STATUS[816].EXT.ModeBit3 := FALSE;
   STATUS[816].EXT.BIT19 := FALSE;
   STATUS[816].EXT.BIT20 := FALSE;
   STATUS[816].EXT.AlarmSuppressed := FALSE;
   STATUS[816].EXT.AlarmPrsent := FALSE;
   STATUS[816].EXT.AlarmFailUnAck := FALSE;
   STATUS[816].Status := 0;
   STATUS[816].TimeStamp := 16#0000;
   STATUS[817].VALUE := 0.0;
   STATUS[817].TRIGVALUE := 0.0;
   STATUS[817].EXT.AlarmWarnUnAck := FALSE;
   STATUS[817].EXT.AckRequired := FALSE;
   STATUS[817].EXT.Maintanence := FALSE;
   STATUS[817].EXT.Operation := FALSE;
   STATUS[817].EXT.Forced := FALSE;
   STATUS[817].EXT.BIT29 := FALSE;
   STATUS[817].EXT.BIT30 := FALSE;
   STATUS[817].EXT.BIT31 := FALSE;
   STATUS[817].EXT.ModeBit1 := FALSE;
   STATUS[817].EXT.ModeBit2 := FALSE;
   STATUS[817].EXT.ModeBit3 := FALSE;
   STATUS[817].EXT.BIT19 := FALSE;
   STATUS[817].EXT.BIT20 := FALSE;
   STATUS[817].EXT.AlarmSuppressed := FALSE;
   STATUS[817].EXT.AlarmPrsent := FALSE;
   STATUS[817].EXT.AlarmFailUnAck := FALSE;
   STATUS[817].Status := 0;
   STATUS[817].TimeStamp := 16#0000;
   STATUS[818].VALUE := 0.0;
   STATUS[818].TRIGVALUE := 0.0;
   STATUS[818].EXT.AlarmWarnUnAck := FALSE;
   STATUS[818].EXT.AckRequired := FALSE;
   STATUS[818].EXT.Maintanence := FALSE;
   STATUS[818].EXT.Operation := FALSE;
   STATUS[818].EXT.Forced := FALSE;
   STATUS[818].EXT.BIT29 := FALSE;
   STATUS[818].EXT.BIT30 := FALSE;
   STATUS[818].EXT.BIT31 := FALSE;
   STATUS[818].EXT.ModeBit1 := FALSE;
   STATUS[818].EXT.ModeBit2 := FALSE;
   STATUS[818].EXT.ModeBit3 := FALSE;
   STATUS[818].EXT.BIT19 := FALSE;
   STATUS[818].EXT.BIT20 := FALSE;
   STATUS[818].EXT.AlarmSuppressed := FALSE;
   STATUS[818].EXT.AlarmPrsent := FALSE;
   STATUS[818].EXT.AlarmFailUnAck := FALSE;
   STATUS[818].Status := 0;
   STATUS[818].TimeStamp := 16#0000;
   STATUS[819].VALUE := 0.0;
   STATUS[819].TRIGVALUE := 0.0;
   STATUS[819].EXT.AlarmWarnUnAck := FALSE;
   STATUS[819].EXT.AckRequired := FALSE;
   STATUS[819].EXT.Maintanence := FALSE;
   STATUS[819].EXT.Operation := FALSE;
   STATUS[819].EXT.Forced := FALSE;
   STATUS[819].EXT.BIT29 := FALSE;
   STATUS[819].EXT.BIT30 := FALSE;
   STATUS[819].EXT.BIT31 := FALSE;
   STATUS[819].EXT.ModeBit1 := FALSE;
   STATUS[819].EXT.ModeBit2 := FALSE;
   STATUS[819].EXT.ModeBit3 := FALSE;
   STATUS[819].EXT.BIT19 := FALSE;
   STATUS[819].EXT.BIT20 := FALSE;
   STATUS[819].EXT.AlarmSuppressed := FALSE;
   STATUS[819].EXT.AlarmPrsent := FALSE;
   STATUS[819].EXT.AlarmFailUnAck := FALSE;
   STATUS[819].Status := 0;
   STATUS[819].TimeStamp := 16#0000;
   STATUS[820].VALUE := 0.0;
   STATUS[820].TRIGVALUE := 0.0;
   STATUS[820].EXT.AlarmWarnUnAck := FALSE;
   STATUS[820].EXT.AckRequired := FALSE;
   STATUS[820].EXT.Maintanence := FALSE;
   STATUS[820].EXT.Operation := FALSE;
   STATUS[820].EXT.Forced := FALSE;
   STATUS[820].EXT.BIT29 := FALSE;
   STATUS[820].EXT.BIT30 := FALSE;
   STATUS[820].EXT.BIT31 := FALSE;
   STATUS[820].EXT.ModeBit1 := FALSE;
   STATUS[820].EXT.ModeBit2 := FALSE;
   STATUS[820].EXT.ModeBit3 := FALSE;
   STATUS[820].EXT.BIT19 := FALSE;
   STATUS[820].EXT.BIT20 := FALSE;
   STATUS[820].EXT.AlarmSuppressed := FALSE;
   STATUS[820].EXT.AlarmPrsent := FALSE;
   STATUS[820].EXT.AlarmFailUnAck := FALSE;
   STATUS[820].Status := 0;
   STATUS[820].TimeStamp := 16#0000;
   STATUS[821].VALUE := 0.0;
   STATUS[821].TRIGVALUE := 0.0;
   STATUS[821].EXT.AlarmWarnUnAck := FALSE;
   STATUS[821].EXT.AckRequired := FALSE;
   STATUS[821].EXT.Maintanence := FALSE;
   STATUS[821].EXT.Operation := FALSE;
   STATUS[821].EXT.Forced := FALSE;
   STATUS[821].EXT.BIT29 := FALSE;
   STATUS[821].EXT.BIT30 := FALSE;
   STATUS[821].EXT.BIT31 := FALSE;
   STATUS[821].EXT.ModeBit1 := FALSE;
   STATUS[821].EXT.ModeBit2 := FALSE;
   STATUS[821].EXT.ModeBit3 := FALSE;
   STATUS[821].EXT.BIT19 := FALSE;
   STATUS[821].EXT.BIT20 := FALSE;
   STATUS[821].EXT.AlarmSuppressed := FALSE;
   STATUS[821].EXT.AlarmPrsent := FALSE;
   STATUS[821].EXT.AlarmFailUnAck := FALSE;
   STATUS[821].Status := 0;
   STATUS[821].TimeStamp := 16#0000;
   STATUS[822].VALUE := 0.0;
   STATUS[822].TRIGVALUE := 0.0;
   STATUS[822].EXT.AlarmWarnUnAck := FALSE;
   STATUS[822].EXT.AckRequired := FALSE;
   STATUS[822].EXT.Maintanence := FALSE;
   STATUS[822].EXT.Operation := FALSE;
   STATUS[822].EXT.Forced := FALSE;
   STATUS[822].EXT.BIT29 := FALSE;
   STATUS[822].EXT.BIT30 := FALSE;
   STATUS[822].EXT.BIT31 := FALSE;
   STATUS[822].EXT.ModeBit1 := FALSE;
   STATUS[822].EXT.ModeBit2 := FALSE;
   STATUS[822].EXT.ModeBit3 := FALSE;
   STATUS[822].EXT.BIT19 := FALSE;
   STATUS[822].EXT.BIT20 := FALSE;
   STATUS[822].EXT.AlarmSuppressed := FALSE;
   STATUS[822].EXT.AlarmPrsent := FALSE;
   STATUS[822].EXT.AlarmFailUnAck := FALSE;
   STATUS[822].Status := 0;
   STATUS[822].TimeStamp := 16#0000;
   STATUS[823].VALUE := 0.0;
   STATUS[823].TRIGVALUE := 0.0;
   STATUS[823].EXT.AlarmWarnUnAck := FALSE;
   STATUS[823].EXT.AckRequired := FALSE;
   STATUS[823].EXT.Maintanence := FALSE;
   STATUS[823].EXT.Operation := FALSE;
   STATUS[823].EXT.Forced := FALSE;
   STATUS[823].EXT.BIT29 := FALSE;
   STATUS[823].EXT.BIT30 := FALSE;
   STATUS[823].EXT.BIT31 := FALSE;
   STATUS[823].EXT.ModeBit1 := FALSE;
   STATUS[823].EXT.ModeBit2 := FALSE;
   STATUS[823].EXT.ModeBit3 := FALSE;
   STATUS[823].EXT.BIT19 := FALSE;
   STATUS[823].EXT.BIT20 := FALSE;
   STATUS[823].EXT.AlarmSuppressed := FALSE;
   STATUS[823].EXT.AlarmPrsent := FALSE;
   STATUS[823].EXT.AlarmFailUnAck := FALSE;
   STATUS[823].Status := 0;
   STATUS[823].TimeStamp := 16#0000;
   STATUS[824].VALUE := 0.0;
   STATUS[824].TRIGVALUE := 0.0;
   STATUS[824].EXT.AlarmWarnUnAck := FALSE;
   STATUS[824].EXT.AckRequired := FALSE;
   STATUS[824].EXT.Maintanence := FALSE;
   STATUS[824].EXT.Operation := FALSE;
   STATUS[824].EXT.Forced := FALSE;
   STATUS[824].EXT.BIT29 := FALSE;
   STATUS[824].EXT.BIT30 := FALSE;
   STATUS[824].EXT.BIT31 := FALSE;
   STATUS[824].EXT.ModeBit1 := FALSE;
   STATUS[824].EXT.ModeBit2 := FALSE;
   STATUS[824].EXT.ModeBit3 := FALSE;
   STATUS[824].EXT.BIT19 := FALSE;
   STATUS[824].EXT.BIT20 := FALSE;
   STATUS[824].EXT.AlarmSuppressed := FALSE;
   STATUS[824].EXT.AlarmPrsent := FALSE;
   STATUS[824].EXT.AlarmFailUnAck := FALSE;
   STATUS[824].Status := 0;
   STATUS[824].TimeStamp := 16#0000;
   STATUS[825].VALUE := 0.0;
   STATUS[825].TRIGVALUE := 0.0;
   STATUS[825].EXT.AlarmWarnUnAck := FALSE;
   STATUS[825].EXT.AckRequired := FALSE;
   STATUS[825].EXT.Maintanence := FALSE;
   STATUS[825].EXT.Operation := FALSE;
   STATUS[825].EXT.Forced := FALSE;
   STATUS[825].EXT.BIT29 := FALSE;
   STATUS[825].EXT.BIT30 := FALSE;
   STATUS[825].EXT.BIT31 := FALSE;
   STATUS[825].EXT.ModeBit1 := FALSE;
   STATUS[825].EXT.ModeBit2 := FALSE;
   STATUS[825].EXT.ModeBit3 := FALSE;
   STATUS[825].EXT.BIT19 := FALSE;
   STATUS[825].EXT.BIT20 := FALSE;
   STATUS[825].EXT.AlarmSuppressed := FALSE;
   STATUS[825].EXT.AlarmPrsent := FALSE;
   STATUS[825].EXT.AlarmFailUnAck := FALSE;
   STATUS[825].Status := 0;
   STATUS[825].TimeStamp := 16#0000;
   STATUS[826].VALUE := 0.0;
   STATUS[826].TRIGVALUE := 0.0;
   STATUS[826].EXT.AlarmWarnUnAck := FALSE;
   STATUS[826].EXT.AckRequired := FALSE;
   STATUS[826].EXT.Maintanence := FALSE;
   STATUS[826].EXT.Operation := FALSE;
   STATUS[826].EXT.Forced := FALSE;
   STATUS[826].EXT.BIT29 := FALSE;
   STATUS[826].EXT.BIT30 := FALSE;
   STATUS[826].EXT.BIT31 := FALSE;
   STATUS[826].EXT.ModeBit1 := FALSE;
   STATUS[826].EXT.ModeBit2 := FALSE;
   STATUS[826].EXT.ModeBit3 := FALSE;
   STATUS[826].EXT.BIT19 := FALSE;
   STATUS[826].EXT.BIT20 := FALSE;
   STATUS[826].EXT.AlarmSuppressed := FALSE;
   STATUS[826].EXT.AlarmPrsent := FALSE;
   STATUS[826].EXT.AlarmFailUnAck := FALSE;
   STATUS[826].Status := 0;
   STATUS[826].TimeStamp := 16#0000;
   STATUS[827].VALUE := 0.0;
   STATUS[827].TRIGVALUE := 0.0;
   STATUS[827].EXT.AlarmWarnUnAck := FALSE;
   STATUS[827].EXT.AckRequired := FALSE;
   STATUS[827].EXT.Maintanence := FALSE;
   STATUS[827].EXT.Operation := FALSE;
   STATUS[827].EXT.Forced := FALSE;
   STATUS[827].EXT.BIT29 := FALSE;
   STATUS[827].EXT.BIT30 := FALSE;
   STATUS[827].EXT.BIT31 := FALSE;
   STATUS[827].EXT.ModeBit1 := FALSE;
   STATUS[827].EXT.ModeBit2 := FALSE;
   STATUS[827].EXT.ModeBit3 := FALSE;
   STATUS[827].EXT.BIT19 := FALSE;
   STATUS[827].EXT.BIT20 := FALSE;
   STATUS[827].EXT.AlarmSuppressed := FALSE;
   STATUS[827].EXT.AlarmPrsent := FALSE;
   STATUS[827].EXT.AlarmFailUnAck := FALSE;
   STATUS[827].Status := 0;
   STATUS[827].TimeStamp := 16#0000;
   STATUS[828].VALUE := 0.0;
   STATUS[828].TRIGVALUE := 0.0;
   STATUS[828].EXT.AlarmWarnUnAck := FALSE;
   STATUS[828].EXT.AckRequired := FALSE;
   STATUS[828].EXT.Maintanence := FALSE;
   STATUS[828].EXT.Operation := FALSE;
   STATUS[828].EXT.Forced := FALSE;
   STATUS[828].EXT.BIT29 := FALSE;
   STATUS[828].EXT.BIT30 := FALSE;
   STATUS[828].EXT.BIT31 := FALSE;
   STATUS[828].EXT.ModeBit1 := FALSE;
   STATUS[828].EXT.ModeBit2 := FALSE;
   STATUS[828].EXT.ModeBit3 := FALSE;
   STATUS[828].EXT.BIT19 := FALSE;
   STATUS[828].EXT.BIT20 := FALSE;
   STATUS[828].EXT.AlarmSuppressed := FALSE;
   STATUS[828].EXT.AlarmPrsent := FALSE;
   STATUS[828].EXT.AlarmFailUnAck := FALSE;
   STATUS[828].Status := 0;
   STATUS[828].TimeStamp := 16#0000;
   STATUS[829].VALUE := 0.0;
   STATUS[829].TRIGVALUE := 0.0;
   STATUS[829].EXT.AlarmWarnUnAck := FALSE;
   STATUS[829].EXT.AckRequired := FALSE;
   STATUS[829].EXT.Maintanence := FALSE;
   STATUS[829].EXT.Operation := FALSE;
   STATUS[829].EXT.Forced := FALSE;
   STATUS[829].EXT.BIT29 := FALSE;
   STATUS[829].EXT.BIT30 := FALSE;
   STATUS[829].EXT.BIT31 := FALSE;
   STATUS[829].EXT.ModeBit1 := FALSE;
   STATUS[829].EXT.ModeBit2 := FALSE;
   STATUS[829].EXT.ModeBit3 := FALSE;
   STATUS[829].EXT.BIT19 := FALSE;
   STATUS[829].EXT.BIT20 := FALSE;
   STATUS[829].EXT.AlarmSuppressed := FALSE;
   STATUS[829].EXT.AlarmPrsent := FALSE;
   STATUS[829].EXT.AlarmFailUnAck := FALSE;
   STATUS[829].Status := 0;
   STATUS[829].TimeStamp := 16#0000;
   STATUS[830].VALUE := 0.0;
   STATUS[830].TRIGVALUE := 0.0;
   STATUS[830].EXT.AlarmWarnUnAck := FALSE;
   STATUS[830].EXT.AckRequired := FALSE;
   STATUS[830].EXT.Maintanence := FALSE;
   STATUS[830].EXT.Operation := FALSE;
   STATUS[830].EXT.Forced := FALSE;
   STATUS[830].EXT.BIT29 := FALSE;
   STATUS[830].EXT.BIT30 := FALSE;
   STATUS[830].EXT.BIT31 := FALSE;
   STATUS[830].EXT.ModeBit1 := FALSE;
   STATUS[830].EXT.ModeBit2 := FALSE;
   STATUS[830].EXT.ModeBit3 := FALSE;
   STATUS[830].EXT.BIT19 := FALSE;
   STATUS[830].EXT.BIT20 := FALSE;
   STATUS[830].EXT.AlarmSuppressed := FALSE;
   STATUS[830].EXT.AlarmPrsent := FALSE;
   STATUS[830].EXT.AlarmFailUnAck := FALSE;
   STATUS[830].Status := 0;
   STATUS[830].TimeStamp := 16#0000;
   STATUS[831].VALUE := 0.0;
   STATUS[831].TRIGVALUE := 0.0;
   STATUS[831].EXT.AlarmWarnUnAck := FALSE;
   STATUS[831].EXT.AckRequired := FALSE;
   STATUS[831].EXT.Maintanence := FALSE;
   STATUS[831].EXT.Operation := FALSE;
   STATUS[831].EXT.Forced := FALSE;
   STATUS[831].EXT.BIT29 := FALSE;
   STATUS[831].EXT.BIT30 := FALSE;
   STATUS[831].EXT.BIT31 := FALSE;
   STATUS[831].EXT.ModeBit1 := FALSE;
   STATUS[831].EXT.ModeBit2 := FALSE;
   STATUS[831].EXT.ModeBit3 := FALSE;
   STATUS[831].EXT.BIT19 := FALSE;
   STATUS[831].EXT.BIT20 := FALSE;
   STATUS[831].EXT.AlarmSuppressed := FALSE;
   STATUS[831].EXT.AlarmPrsent := FALSE;
   STATUS[831].EXT.AlarmFailUnAck := FALSE;
   STATUS[831].Status := 0;
   STATUS[831].TimeStamp := 16#0000;
   STATUS[832].VALUE := 0.0;
   STATUS[832].TRIGVALUE := 0.0;
   STATUS[832].EXT.AlarmWarnUnAck := FALSE;
   STATUS[832].EXT.AckRequired := FALSE;
   STATUS[832].EXT.Maintanence := FALSE;
   STATUS[832].EXT.Operation := FALSE;
   STATUS[832].EXT.Forced := FALSE;
   STATUS[832].EXT.BIT29 := FALSE;
   STATUS[832].EXT.BIT30 := FALSE;
   STATUS[832].EXT.BIT31 := FALSE;
   STATUS[832].EXT.ModeBit1 := FALSE;
   STATUS[832].EXT.ModeBit2 := FALSE;
   STATUS[832].EXT.ModeBit3 := FALSE;
   STATUS[832].EXT.BIT19 := FALSE;
   STATUS[832].EXT.BIT20 := FALSE;
   STATUS[832].EXT.AlarmSuppressed := FALSE;
   STATUS[832].EXT.AlarmPrsent := FALSE;
   STATUS[832].EXT.AlarmFailUnAck := FALSE;
   STATUS[832].Status := 0;
   STATUS[832].TimeStamp := 16#0000;
   STATUS[833].VALUE := 0.0;
   STATUS[833].TRIGVALUE := 0.0;
   STATUS[833].EXT.AlarmWarnUnAck := FALSE;
   STATUS[833].EXT.AckRequired := FALSE;
   STATUS[833].EXT.Maintanence := FALSE;
   STATUS[833].EXT.Operation := FALSE;
   STATUS[833].EXT.Forced := FALSE;
   STATUS[833].EXT.BIT29 := FALSE;
   STATUS[833].EXT.BIT30 := FALSE;
   STATUS[833].EXT.BIT31 := FALSE;
   STATUS[833].EXT.ModeBit1 := FALSE;
   STATUS[833].EXT.ModeBit2 := FALSE;
   STATUS[833].EXT.ModeBit3 := FALSE;
   STATUS[833].EXT.BIT19 := FALSE;
   STATUS[833].EXT.BIT20 := FALSE;
   STATUS[833].EXT.AlarmSuppressed := FALSE;
   STATUS[833].EXT.AlarmPrsent := FALSE;
   STATUS[833].EXT.AlarmFailUnAck := FALSE;
   STATUS[833].Status := 0;
   STATUS[833].TimeStamp := 16#0000;
   STATUS[834].VALUE := 0.0;
   STATUS[834].TRIGVALUE := 0.0;
   STATUS[834].EXT.AlarmWarnUnAck := FALSE;
   STATUS[834].EXT.AckRequired := FALSE;
   STATUS[834].EXT.Maintanence := FALSE;
   STATUS[834].EXT.Operation := FALSE;
   STATUS[834].EXT.Forced := FALSE;
   STATUS[834].EXT.BIT29 := FALSE;
   STATUS[834].EXT.BIT30 := FALSE;
   STATUS[834].EXT.BIT31 := FALSE;
   STATUS[834].EXT.ModeBit1 := FALSE;
   STATUS[834].EXT.ModeBit2 := FALSE;
   STATUS[834].EXT.ModeBit3 := FALSE;
   STATUS[834].EXT.BIT19 := FALSE;
   STATUS[834].EXT.BIT20 := FALSE;
   STATUS[834].EXT.AlarmSuppressed := FALSE;
   STATUS[834].EXT.AlarmPrsent := FALSE;
   STATUS[834].EXT.AlarmFailUnAck := FALSE;
   STATUS[834].Status := 0;
   STATUS[834].TimeStamp := 16#0000;
   STATUS[835].VALUE := 0.0;
   STATUS[835].TRIGVALUE := 0.0;
   STATUS[835].EXT.AlarmWarnUnAck := FALSE;
   STATUS[835].EXT.AckRequired := FALSE;
   STATUS[835].EXT.Maintanence := FALSE;
   STATUS[835].EXT.Operation := FALSE;
   STATUS[835].EXT.Forced := FALSE;
   STATUS[835].EXT.BIT29 := FALSE;
   STATUS[835].EXT.BIT30 := FALSE;
   STATUS[835].EXT.BIT31 := FALSE;
   STATUS[835].EXT.ModeBit1 := FALSE;
   STATUS[835].EXT.ModeBit2 := FALSE;
   STATUS[835].EXT.ModeBit3 := FALSE;
   STATUS[835].EXT.BIT19 := FALSE;
   STATUS[835].EXT.BIT20 := FALSE;
   STATUS[835].EXT.AlarmSuppressed := FALSE;
   STATUS[835].EXT.AlarmPrsent := FALSE;
   STATUS[835].EXT.AlarmFailUnAck := FALSE;
   STATUS[835].Status := 0;
   STATUS[835].TimeStamp := 16#0000;
   STATUS[836].VALUE := 0.0;
   STATUS[836].TRIGVALUE := 0.0;
   STATUS[836].EXT.AlarmWarnUnAck := FALSE;
   STATUS[836].EXT.AckRequired := FALSE;
   STATUS[836].EXT.Maintanence := FALSE;
   STATUS[836].EXT.Operation := FALSE;
   STATUS[836].EXT.Forced := FALSE;
   STATUS[836].EXT.BIT29 := FALSE;
   STATUS[836].EXT.BIT30 := FALSE;
   STATUS[836].EXT.BIT31 := FALSE;
   STATUS[836].EXT.ModeBit1 := FALSE;
   STATUS[836].EXT.ModeBit2 := FALSE;
   STATUS[836].EXT.ModeBit3 := FALSE;
   STATUS[836].EXT.BIT19 := FALSE;
   STATUS[836].EXT.BIT20 := FALSE;
   STATUS[836].EXT.AlarmSuppressed := FALSE;
   STATUS[836].EXT.AlarmPrsent := FALSE;
   STATUS[836].EXT.AlarmFailUnAck := FALSE;
   STATUS[836].Status := 0;
   STATUS[836].TimeStamp := 16#0000;
   STATUS[837].VALUE := 0.0;
   STATUS[837].TRIGVALUE := 0.0;
   STATUS[837].EXT.AlarmWarnUnAck := FALSE;
   STATUS[837].EXT.AckRequired := FALSE;
   STATUS[837].EXT.Maintanence := FALSE;
   STATUS[837].EXT.Operation := FALSE;
   STATUS[837].EXT.Forced := FALSE;
   STATUS[837].EXT.BIT29 := FALSE;
   STATUS[837].EXT.BIT30 := FALSE;
   STATUS[837].EXT.BIT31 := FALSE;
   STATUS[837].EXT.ModeBit1 := FALSE;
   STATUS[837].EXT.ModeBit2 := FALSE;
   STATUS[837].EXT.ModeBit3 := FALSE;
   STATUS[837].EXT.BIT19 := FALSE;
   STATUS[837].EXT.BIT20 := FALSE;
   STATUS[837].EXT.AlarmSuppressed := FALSE;
   STATUS[837].EXT.AlarmPrsent := FALSE;
   STATUS[837].EXT.AlarmFailUnAck := FALSE;
   STATUS[837].Status := 0;
   STATUS[837].TimeStamp := 16#0000;
   STATUS[838].VALUE := 0.0;
   STATUS[838].TRIGVALUE := 0.0;
   STATUS[838].EXT.AlarmWarnUnAck := FALSE;
   STATUS[838].EXT.AckRequired := FALSE;
   STATUS[838].EXT.Maintanence := FALSE;
   STATUS[838].EXT.Operation := FALSE;
   STATUS[838].EXT.Forced := FALSE;
   STATUS[838].EXT.BIT29 := FALSE;
   STATUS[838].EXT.BIT30 := FALSE;
   STATUS[838].EXT.BIT31 := FALSE;
   STATUS[838].EXT.ModeBit1 := FALSE;
   STATUS[838].EXT.ModeBit2 := FALSE;
   STATUS[838].EXT.ModeBit3 := FALSE;
   STATUS[838].EXT.BIT19 := FALSE;
   STATUS[838].EXT.BIT20 := FALSE;
   STATUS[838].EXT.AlarmSuppressed := FALSE;
   STATUS[838].EXT.AlarmPrsent := FALSE;
   STATUS[838].EXT.AlarmFailUnAck := FALSE;
   STATUS[838].Status := 0;
   STATUS[838].TimeStamp := 16#0000;
   STATUS[839].VALUE := 0.0;
   STATUS[839].TRIGVALUE := 0.0;
   STATUS[839].EXT.AlarmWarnUnAck := FALSE;
   STATUS[839].EXT.AckRequired := FALSE;
   STATUS[839].EXT.Maintanence := FALSE;
   STATUS[839].EXT.Operation := FALSE;
   STATUS[839].EXT.Forced := FALSE;
   STATUS[839].EXT.BIT29 := FALSE;
   STATUS[839].EXT.BIT30 := FALSE;
   STATUS[839].EXT.BIT31 := FALSE;
   STATUS[839].EXT.ModeBit1 := FALSE;
   STATUS[839].EXT.ModeBit2 := FALSE;
   STATUS[839].EXT.ModeBit3 := FALSE;
   STATUS[839].EXT.BIT19 := FALSE;
   STATUS[839].EXT.BIT20 := FALSE;
   STATUS[839].EXT.AlarmSuppressed := FALSE;
   STATUS[839].EXT.AlarmPrsent := FALSE;
   STATUS[839].EXT.AlarmFailUnAck := FALSE;
   STATUS[839].Status := 0;
   STATUS[839].TimeStamp := 16#0000;
   STATUS[840].VALUE := 0.0;
   STATUS[840].TRIGVALUE := 0.0;
   STATUS[840].EXT.AlarmWarnUnAck := FALSE;
   STATUS[840].EXT.AckRequired := FALSE;
   STATUS[840].EXT.Maintanence := FALSE;
   STATUS[840].EXT.Operation := FALSE;
   STATUS[840].EXT.Forced := FALSE;
   STATUS[840].EXT.BIT29 := FALSE;
   STATUS[840].EXT.BIT30 := FALSE;
   STATUS[840].EXT.BIT31 := FALSE;
   STATUS[840].EXT.ModeBit1 := FALSE;
   STATUS[840].EXT.ModeBit2 := FALSE;
   STATUS[840].EXT.ModeBit3 := FALSE;
   STATUS[840].EXT.BIT19 := FALSE;
   STATUS[840].EXT.BIT20 := FALSE;
   STATUS[840].EXT.AlarmSuppressed := FALSE;
   STATUS[840].EXT.AlarmPrsent := FALSE;
   STATUS[840].EXT.AlarmFailUnAck := FALSE;
   STATUS[840].Status := 0;
   STATUS[840].TimeStamp := 16#0000;
   STATUS[841].VALUE := 0.0;
   STATUS[841].TRIGVALUE := 0.0;
   STATUS[841].EXT.AlarmWarnUnAck := FALSE;
   STATUS[841].EXT.AckRequired := FALSE;
   STATUS[841].EXT.Maintanence := FALSE;
   STATUS[841].EXT.Operation := FALSE;
   STATUS[841].EXT.Forced := FALSE;
   STATUS[841].EXT.BIT29 := FALSE;
   STATUS[841].EXT.BIT30 := FALSE;
   STATUS[841].EXT.BIT31 := FALSE;
   STATUS[841].EXT.ModeBit1 := FALSE;
   STATUS[841].EXT.ModeBit2 := FALSE;
   STATUS[841].EXT.ModeBit3 := FALSE;
   STATUS[841].EXT.BIT19 := FALSE;
   STATUS[841].EXT.BIT20 := FALSE;
   STATUS[841].EXT.AlarmSuppressed := FALSE;
   STATUS[841].EXT.AlarmPrsent := FALSE;
   STATUS[841].EXT.AlarmFailUnAck := FALSE;
   STATUS[841].Status := 0;
   STATUS[841].TimeStamp := 16#0000;
   STATUS[842].VALUE := 0.0;
   STATUS[842].TRIGVALUE := 0.0;
   STATUS[842].EXT.AlarmWarnUnAck := FALSE;
   STATUS[842].EXT.AckRequired := FALSE;
   STATUS[842].EXT.Maintanence := FALSE;
   STATUS[842].EXT.Operation := FALSE;
   STATUS[842].EXT.Forced := FALSE;
   STATUS[842].EXT.BIT29 := FALSE;
   STATUS[842].EXT.BIT30 := FALSE;
   STATUS[842].EXT.BIT31 := FALSE;
   STATUS[842].EXT.ModeBit1 := FALSE;
   STATUS[842].EXT.ModeBit2 := FALSE;
   STATUS[842].EXT.ModeBit3 := FALSE;
   STATUS[842].EXT.BIT19 := FALSE;
   STATUS[842].EXT.BIT20 := FALSE;
   STATUS[842].EXT.AlarmSuppressed := FALSE;
   STATUS[842].EXT.AlarmPrsent := FALSE;
   STATUS[842].EXT.AlarmFailUnAck := FALSE;
   STATUS[842].Status := 0;
   STATUS[842].TimeStamp := 16#0000;
   STATUS[843].VALUE := 0.0;
   STATUS[843].TRIGVALUE := 0.0;
   STATUS[843].EXT.AlarmWarnUnAck := FALSE;
   STATUS[843].EXT.AckRequired := FALSE;
   STATUS[843].EXT.Maintanence := FALSE;
   STATUS[843].EXT.Operation := FALSE;
   STATUS[843].EXT.Forced := FALSE;
   STATUS[843].EXT.BIT29 := FALSE;
   STATUS[843].EXT.BIT30 := FALSE;
   STATUS[843].EXT.BIT31 := FALSE;
   STATUS[843].EXT.ModeBit1 := FALSE;
   STATUS[843].EXT.ModeBit2 := FALSE;
   STATUS[843].EXT.ModeBit3 := FALSE;
   STATUS[843].EXT.BIT19 := FALSE;
   STATUS[843].EXT.BIT20 := FALSE;
   STATUS[843].EXT.AlarmSuppressed := FALSE;
   STATUS[843].EXT.AlarmPrsent := FALSE;
   STATUS[843].EXT.AlarmFailUnAck := FALSE;
   STATUS[843].Status := 0;
   STATUS[843].TimeStamp := 16#0000;
   STATUS[844].VALUE := 0.0;
   STATUS[844].TRIGVALUE := 0.0;
   STATUS[844].EXT.AlarmWarnUnAck := FALSE;
   STATUS[844].EXT.AckRequired := FALSE;
   STATUS[844].EXT.Maintanence := FALSE;
   STATUS[844].EXT.Operation := FALSE;
   STATUS[844].EXT.Forced := FALSE;
   STATUS[844].EXT.BIT29 := FALSE;
   STATUS[844].EXT.BIT30 := FALSE;
   STATUS[844].EXT.BIT31 := FALSE;
   STATUS[844].EXT.ModeBit1 := FALSE;
   STATUS[844].EXT.ModeBit2 := FALSE;
   STATUS[844].EXT.ModeBit3 := FALSE;
   STATUS[844].EXT.BIT19 := FALSE;
   STATUS[844].EXT.BIT20 := FALSE;
   STATUS[844].EXT.AlarmSuppressed := FALSE;
   STATUS[844].EXT.AlarmPrsent := FALSE;
   STATUS[844].EXT.AlarmFailUnAck := FALSE;
   STATUS[844].Status := 0;
   STATUS[844].TimeStamp := 16#0000;
   STATUS[845].VALUE := 0.0;
   STATUS[845].TRIGVALUE := 0.0;
   STATUS[845].EXT.AlarmWarnUnAck := FALSE;
   STATUS[845].EXT.AckRequired := FALSE;
   STATUS[845].EXT.Maintanence := FALSE;
   STATUS[845].EXT.Operation := FALSE;
   STATUS[845].EXT.Forced := FALSE;
   STATUS[845].EXT.BIT29 := FALSE;
   STATUS[845].EXT.BIT30 := FALSE;
   STATUS[845].EXT.BIT31 := FALSE;
   STATUS[845].EXT.ModeBit1 := FALSE;
   STATUS[845].EXT.ModeBit2 := FALSE;
   STATUS[845].EXT.ModeBit3 := FALSE;
   STATUS[845].EXT.BIT19 := FALSE;
   STATUS[845].EXT.BIT20 := FALSE;
   STATUS[845].EXT.AlarmSuppressed := FALSE;
   STATUS[845].EXT.AlarmPrsent := FALSE;
   STATUS[845].EXT.AlarmFailUnAck := FALSE;
   STATUS[845].Status := 0;
   STATUS[845].TimeStamp := 16#0000;
   STATUS[846].VALUE := 0.0;
   STATUS[846].TRIGVALUE := 0.0;
   STATUS[846].EXT.AlarmWarnUnAck := FALSE;
   STATUS[846].EXT.AckRequired := FALSE;
   STATUS[846].EXT.Maintanence := FALSE;
   STATUS[846].EXT.Operation := FALSE;
   STATUS[846].EXT.Forced := FALSE;
   STATUS[846].EXT.BIT29 := FALSE;
   STATUS[846].EXT.BIT30 := FALSE;
   STATUS[846].EXT.BIT31 := FALSE;
   STATUS[846].EXT.ModeBit1 := FALSE;
   STATUS[846].EXT.ModeBit2 := FALSE;
   STATUS[846].EXT.ModeBit3 := FALSE;
   STATUS[846].EXT.BIT19 := FALSE;
   STATUS[846].EXT.BIT20 := FALSE;
   STATUS[846].EXT.AlarmSuppressed := FALSE;
   STATUS[846].EXT.AlarmPrsent := FALSE;
   STATUS[846].EXT.AlarmFailUnAck := FALSE;
   STATUS[846].Status := 0;
   STATUS[846].TimeStamp := 16#0000;
   STATUS[847].VALUE := 0.0;
   STATUS[847].TRIGVALUE := 0.0;
   STATUS[847].EXT.AlarmWarnUnAck := FALSE;
   STATUS[847].EXT.AckRequired := FALSE;
   STATUS[847].EXT.Maintanence := FALSE;
   STATUS[847].EXT.Operation := FALSE;
   STATUS[847].EXT.Forced := FALSE;
   STATUS[847].EXT.BIT29 := FALSE;
   STATUS[847].EXT.BIT30 := FALSE;
   STATUS[847].EXT.BIT31 := FALSE;
   STATUS[847].EXT.ModeBit1 := FALSE;
   STATUS[847].EXT.ModeBit2 := FALSE;
   STATUS[847].EXT.ModeBit3 := FALSE;
   STATUS[847].EXT.BIT19 := FALSE;
   STATUS[847].EXT.BIT20 := FALSE;
   STATUS[847].EXT.AlarmSuppressed := FALSE;
   STATUS[847].EXT.AlarmPrsent := FALSE;
   STATUS[847].EXT.AlarmFailUnAck := FALSE;
   STATUS[847].Status := 0;
   STATUS[847].TimeStamp := 16#0000;
   STATUS[848].VALUE := 0.0;
   STATUS[848].TRIGVALUE := 0.0;
   STATUS[848].EXT.AlarmWarnUnAck := FALSE;
   STATUS[848].EXT.AckRequired := FALSE;
   STATUS[848].EXT.Maintanence := FALSE;
   STATUS[848].EXT.Operation := FALSE;
   STATUS[848].EXT.Forced := FALSE;
   STATUS[848].EXT.BIT29 := FALSE;
   STATUS[848].EXT.BIT30 := FALSE;
   STATUS[848].EXT.BIT31 := FALSE;
   STATUS[848].EXT.ModeBit1 := FALSE;
   STATUS[848].EXT.ModeBit2 := FALSE;
   STATUS[848].EXT.ModeBit3 := FALSE;
   STATUS[848].EXT.BIT19 := FALSE;
   STATUS[848].EXT.BIT20 := FALSE;
   STATUS[848].EXT.AlarmSuppressed := FALSE;
   STATUS[848].EXT.AlarmPrsent := FALSE;
   STATUS[848].EXT.AlarmFailUnAck := FALSE;
   STATUS[848].Status := 0;
   STATUS[848].TimeStamp := 16#0000;
   STATUS[849].VALUE := 0.0;
   STATUS[849].TRIGVALUE := 0.0;
   STATUS[849].EXT.AlarmWarnUnAck := FALSE;
   STATUS[849].EXT.AckRequired := FALSE;
   STATUS[849].EXT.Maintanence := FALSE;
   STATUS[849].EXT.Operation := FALSE;
   STATUS[849].EXT.Forced := FALSE;
   STATUS[849].EXT.BIT29 := FALSE;
   STATUS[849].EXT.BIT30 := FALSE;
   STATUS[849].EXT.BIT31 := FALSE;
   STATUS[849].EXT.ModeBit1 := FALSE;
   STATUS[849].EXT.ModeBit2 := FALSE;
   STATUS[849].EXT.ModeBit3 := FALSE;
   STATUS[849].EXT.BIT19 := FALSE;
   STATUS[849].EXT.BIT20 := FALSE;
   STATUS[849].EXT.AlarmSuppressed := FALSE;
   STATUS[849].EXT.AlarmPrsent := FALSE;
   STATUS[849].EXT.AlarmFailUnAck := FALSE;
   STATUS[849].Status := 0;
   STATUS[849].TimeStamp := 16#0000;
   STATUS[850].VALUE := 0.0;
   STATUS[850].TRIGVALUE := 0.0;
   STATUS[850].EXT.AlarmWarnUnAck := FALSE;
   STATUS[850].EXT.AckRequired := FALSE;
   STATUS[850].EXT.Maintanence := FALSE;
   STATUS[850].EXT.Operation := FALSE;
   STATUS[850].EXT.Forced := FALSE;
   STATUS[850].EXT.BIT29 := FALSE;
   STATUS[850].EXT.BIT30 := FALSE;
   STATUS[850].EXT.BIT31 := FALSE;
   STATUS[850].EXT.ModeBit1 := FALSE;
   STATUS[850].EXT.ModeBit2 := FALSE;
   STATUS[850].EXT.ModeBit3 := FALSE;
   STATUS[850].EXT.BIT19 := FALSE;
   STATUS[850].EXT.BIT20 := FALSE;
   STATUS[850].EXT.AlarmSuppressed := FALSE;
   STATUS[850].EXT.AlarmPrsent := FALSE;
   STATUS[850].EXT.AlarmFailUnAck := FALSE;
   STATUS[850].Status := 0;
   STATUS[850].TimeStamp := 16#0000;
   STATUS[851].VALUE := 0.0;
   STATUS[851].TRIGVALUE := 0.0;
   STATUS[851].EXT.AlarmWarnUnAck := FALSE;
   STATUS[851].EXT.AckRequired := FALSE;
   STATUS[851].EXT.Maintanence := FALSE;
   STATUS[851].EXT.Operation := FALSE;
   STATUS[851].EXT.Forced := FALSE;
   STATUS[851].EXT.BIT29 := FALSE;
   STATUS[851].EXT.BIT30 := FALSE;
   STATUS[851].EXT.BIT31 := FALSE;
   STATUS[851].EXT.ModeBit1 := FALSE;
   STATUS[851].EXT.ModeBit2 := FALSE;
   STATUS[851].EXT.ModeBit3 := FALSE;
   STATUS[851].EXT.BIT19 := FALSE;
   STATUS[851].EXT.BIT20 := FALSE;
   STATUS[851].EXT.AlarmSuppressed := FALSE;
   STATUS[851].EXT.AlarmPrsent := FALSE;
   STATUS[851].EXT.AlarmFailUnAck := FALSE;
   STATUS[851].Status := 0;
   STATUS[851].TimeStamp := 16#0000;
   STATUS[852].VALUE := 0.0;
   STATUS[852].TRIGVALUE := 0.0;
   STATUS[852].EXT.AlarmWarnUnAck := FALSE;
   STATUS[852].EXT.AckRequired := FALSE;
   STATUS[852].EXT.Maintanence := FALSE;
   STATUS[852].EXT.Operation := FALSE;
   STATUS[852].EXT.Forced := FALSE;
   STATUS[852].EXT.BIT29 := FALSE;
   STATUS[852].EXT.BIT30 := FALSE;
   STATUS[852].EXT.BIT31 := FALSE;
   STATUS[852].EXT.ModeBit1 := FALSE;
   STATUS[852].EXT.ModeBit2 := FALSE;
   STATUS[852].EXT.ModeBit3 := FALSE;
   STATUS[852].EXT.BIT19 := FALSE;
   STATUS[852].EXT.BIT20 := FALSE;
   STATUS[852].EXT.AlarmSuppressed := FALSE;
   STATUS[852].EXT.AlarmPrsent := FALSE;
   STATUS[852].EXT.AlarmFailUnAck := FALSE;
   STATUS[852].Status := 0;
   STATUS[852].TimeStamp := 16#0000;
   STATUS[853].VALUE := 0.0;
   STATUS[853].TRIGVALUE := 0.0;
   STATUS[853].EXT.AlarmWarnUnAck := FALSE;
   STATUS[853].EXT.AckRequired := FALSE;
   STATUS[853].EXT.Maintanence := FALSE;
   STATUS[853].EXT.Operation := FALSE;
   STATUS[853].EXT.Forced := FALSE;
   STATUS[853].EXT.BIT29 := FALSE;
   STATUS[853].EXT.BIT30 := FALSE;
   STATUS[853].EXT.BIT31 := FALSE;
   STATUS[853].EXT.ModeBit1 := FALSE;
   STATUS[853].EXT.ModeBit2 := FALSE;
   STATUS[853].EXT.ModeBit3 := FALSE;
   STATUS[853].EXT.BIT19 := FALSE;
   STATUS[853].EXT.BIT20 := FALSE;
   STATUS[853].EXT.AlarmSuppressed := FALSE;
   STATUS[853].EXT.AlarmPrsent := FALSE;
   STATUS[853].EXT.AlarmFailUnAck := FALSE;
   STATUS[853].Status := 0;
   STATUS[853].TimeStamp := 16#0000;
   STATUS[854].VALUE := 0.0;
   STATUS[854].TRIGVALUE := 0.0;
   STATUS[854].EXT.AlarmWarnUnAck := FALSE;
   STATUS[854].EXT.AckRequired := FALSE;
   STATUS[854].EXT.Maintanence := FALSE;
   STATUS[854].EXT.Operation := FALSE;
   STATUS[854].EXT.Forced := FALSE;
   STATUS[854].EXT.BIT29 := FALSE;
   STATUS[854].EXT.BIT30 := FALSE;
   STATUS[854].EXT.BIT31 := FALSE;
   STATUS[854].EXT.ModeBit1 := FALSE;
   STATUS[854].EXT.ModeBit2 := FALSE;
   STATUS[854].EXT.ModeBit3 := FALSE;
   STATUS[854].EXT.BIT19 := FALSE;
   STATUS[854].EXT.BIT20 := FALSE;
   STATUS[854].EXT.AlarmSuppressed := FALSE;
   STATUS[854].EXT.AlarmPrsent := FALSE;
   STATUS[854].EXT.AlarmFailUnAck := FALSE;
   STATUS[854].Status := 0;
   STATUS[854].TimeStamp := 16#0000;
   STATUS[855].VALUE := 0.0;
   STATUS[855].TRIGVALUE := 0.0;
   STATUS[855].EXT.AlarmWarnUnAck := FALSE;
   STATUS[855].EXT.AckRequired := FALSE;
   STATUS[855].EXT.Maintanence := FALSE;
   STATUS[855].EXT.Operation := FALSE;
   STATUS[855].EXT.Forced := FALSE;
   STATUS[855].EXT.BIT29 := FALSE;
   STATUS[855].EXT.BIT30 := FALSE;
   STATUS[855].EXT.BIT31 := FALSE;
   STATUS[855].EXT.ModeBit1 := FALSE;
   STATUS[855].EXT.ModeBit2 := FALSE;
   STATUS[855].EXT.ModeBit3 := FALSE;
   STATUS[855].EXT.BIT19 := FALSE;
   STATUS[855].EXT.BIT20 := FALSE;
   STATUS[855].EXT.AlarmSuppressed := FALSE;
   STATUS[855].EXT.AlarmPrsent := FALSE;
   STATUS[855].EXT.AlarmFailUnAck := FALSE;
   STATUS[855].Status := 0;
   STATUS[855].TimeStamp := 16#0000;
   STATUS[856].VALUE := 0.0;
   STATUS[856].TRIGVALUE := 0.0;
   STATUS[856].EXT.AlarmWarnUnAck := FALSE;
   STATUS[856].EXT.AckRequired := FALSE;
   STATUS[856].EXT.Maintanence := FALSE;
   STATUS[856].EXT.Operation := FALSE;
   STATUS[856].EXT.Forced := FALSE;
   STATUS[856].EXT.BIT29 := FALSE;
   STATUS[856].EXT.BIT30 := FALSE;
   STATUS[856].EXT.BIT31 := FALSE;
   STATUS[856].EXT.ModeBit1 := FALSE;
   STATUS[856].EXT.ModeBit2 := FALSE;
   STATUS[856].EXT.ModeBit3 := FALSE;
   STATUS[856].EXT.BIT19 := FALSE;
   STATUS[856].EXT.BIT20 := FALSE;
   STATUS[856].EXT.AlarmSuppressed := FALSE;
   STATUS[856].EXT.AlarmPrsent := FALSE;
   STATUS[856].EXT.AlarmFailUnAck := FALSE;
   STATUS[856].Status := 0;
   STATUS[856].TimeStamp := 16#0000;
   STATUS[857].VALUE := 0.0;
   STATUS[857].TRIGVALUE := 0.0;
   STATUS[857].EXT.AlarmWarnUnAck := FALSE;
   STATUS[857].EXT.AckRequired := FALSE;
   STATUS[857].EXT.Maintanence := FALSE;
   STATUS[857].EXT.Operation := FALSE;
   STATUS[857].EXT.Forced := FALSE;
   STATUS[857].EXT.BIT29 := FALSE;
   STATUS[857].EXT.BIT30 := FALSE;
   STATUS[857].EXT.BIT31 := FALSE;
   STATUS[857].EXT.ModeBit1 := FALSE;
   STATUS[857].EXT.ModeBit2 := FALSE;
   STATUS[857].EXT.ModeBit3 := FALSE;
   STATUS[857].EXT.BIT19 := FALSE;
   STATUS[857].EXT.BIT20 := FALSE;
   STATUS[857].EXT.AlarmSuppressed := FALSE;
   STATUS[857].EXT.AlarmPrsent := FALSE;
   STATUS[857].EXT.AlarmFailUnAck := FALSE;
   STATUS[857].Status := 0;
   STATUS[857].TimeStamp := 16#0000;
   STATUS[858].VALUE := 0.0;
   STATUS[858].TRIGVALUE := 0.0;
   STATUS[858].EXT.AlarmWarnUnAck := FALSE;
   STATUS[858].EXT.AckRequired := FALSE;
   STATUS[858].EXT.Maintanence := FALSE;
   STATUS[858].EXT.Operation := FALSE;
   STATUS[858].EXT.Forced := FALSE;
   STATUS[858].EXT.BIT29 := FALSE;
   STATUS[858].EXT.BIT30 := FALSE;
   STATUS[858].EXT.BIT31 := FALSE;
   STATUS[858].EXT.ModeBit1 := FALSE;
   STATUS[858].EXT.ModeBit2 := FALSE;
   STATUS[858].EXT.ModeBit3 := FALSE;
   STATUS[858].EXT.BIT19 := FALSE;
   STATUS[858].EXT.BIT20 := FALSE;
   STATUS[858].EXT.AlarmSuppressed := FALSE;
   STATUS[858].EXT.AlarmPrsent := FALSE;
   STATUS[858].EXT.AlarmFailUnAck := FALSE;
   STATUS[858].Status := 0;
   STATUS[858].TimeStamp := 16#0000;
   STATUS[859].VALUE := 0.0;
   STATUS[859].TRIGVALUE := 0.0;
   STATUS[859].EXT.AlarmWarnUnAck := FALSE;
   STATUS[859].EXT.AckRequired := FALSE;
   STATUS[859].EXT.Maintanence := FALSE;
   STATUS[859].EXT.Operation := FALSE;
   STATUS[859].EXT.Forced := FALSE;
   STATUS[859].EXT.BIT29 := FALSE;
   STATUS[859].EXT.BIT30 := FALSE;
   STATUS[859].EXT.BIT31 := FALSE;
   STATUS[859].EXT.ModeBit1 := FALSE;
   STATUS[859].EXT.ModeBit2 := FALSE;
   STATUS[859].EXT.ModeBit3 := FALSE;
   STATUS[859].EXT.BIT19 := FALSE;
   STATUS[859].EXT.BIT20 := FALSE;
   STATUS[859].EXT.AlarmSuppressed := FALSE;
   STATUS[859].EXT.AlarmPrsent := FALSE;
   STATUS[859].EXT.AlarmFailUnAck := FALSE;
   STATUS[859].Status := 0;
   STATUS[859].TimeStamp := 16#0000;
   STATUS[860].VALUE := 0.0;
   STATUS[860].TRIGVALUE := 0.0;
   STATUS[860].EXT.AlarmWarnUnAck := FALSE;
   STATUS[860].EXT.AckRequired := FALSE;
   STATUS[860].EXT.Maintanence := FALSE;
   STATUS[860].EXT.Operation := FALSE;
   STATUS[860].EXT.Forced := FALSE;
   STATUS[860].EXT.BIT29 := FALSE;
   STATUS[860].EXT.BIT30 := FALSE;
   STATUS[860].EXT.BIT31 := FALSE;
   STATUS[860].EXT.ModeBit1 := FALSE;
   STATUS[860].EXT.ModeBit2 := FALSE;
   STATUS[860].EXT.ModeBit3 := FALSE;
   STATUS[860].EXT.BIT19 := FALSE;
   STATUS[860].EXT.BIT20 := FALSE;
   STATUS[860].EXT.AlarmSuppressed := FALSE;
   STATUS[860].EXT.AlarmPrsent := FALSE;
   STATUS[860].EXT.AlarmFailUnAck := FALSE;
   STATUS[860].Status := 0;
   STATUS[860].TimeStamp := 16#0000;
   STATUS[861].VALUE := 0.0;
   STATUS[861].TRIGVALUE := 0.0;
   STATUS[861].EXT.AlarmWarnUnAck := FALSE;
   STATUS[861].EXT.AckRequired := FALSE;
   STATUS[861].EXT.Maintanence := FALSE;
   STATUS[861].EXT.Operation := FALSE;
   STATUS[861].EXT.Forced := FALSE;
   STATUS[861].EXT.BIT29 := FALSE;
   STATUS[861].EXT.BIT30 := FALSE;
   STATUS[861].EXT.BIT31 := FALSE;
   STATUS[861].EXT.ModeBit1 := FALSE;
   STATUS[861].EXT.ModeBit2 := FALSE;
   STATUS[861].EXT.ModeBit3 := FALSE;
   STATUS[861].EXT.BIT19 := FALSE;
   STATUS[861].EXT.BIT20 := FALSE;
   STATUS[861].EXT.AlarmSuppressed := FALSE;
   STATUS[861].EXT.AlarmPrsent := FALSE;
   STATUS[861].EXT.AlarmFailUnAck := FALSE;
   STATUS[861].Status := 0;
   STATUS[861].TimeStamp := 16#0000;
   STATUS[862].VALUE := 0.0;
   STATUS[862].TRIGVALUE := 0.0;
   STATUS[862].EXT.AlarmWarnUnAck := FALSE;
   STATUS[862].EXT.AckRequired := FALSE;
   STATUS[862].EXT.Maintanence := FALSE;
   STATUS[862].EXT.Operation := FALSE;
   STATUS[862].EXT.Forced := FALSE;
   STATUS[862].EXT.BIT29 := FALSE;
   STATUS[862].EXT.BIT30 := FALSE;
   STATUS[862].EXT.BIT31 := FALSE;
   STATUS[862].EXT.ModeBit1 := FALSE;
   STATUS[862].EXT.ModeBit2 := FALSE;
   STATUS[862].EXT.ModeBit3 := FALSE;
   STATUS[862].EXT.BIT19 := FALSE;
   STATUS[862].EXT.BIT20 := FALSE;
   STATUS[862].EXT.AlarmSuppressed := FALSE;
   STATUS[862].EXT.AlarmPrsent := FALSE;
   STATUS[862].EXT.AlarmFailUnAck := FALSE;
   STATUS[862].Status := 0;
   STATUS[862].TimeStamp := 16#0000;
   STATUS[863].VALUE := 0.0;
   STATUS[863].TRIGVALUE := 0.0;
   STATUS[863].EXT.AlarmWarnUnAck := FALSE;
   STATUS[863].EXT.AckRequired := FALSE;
   STATUS[863].EXT.Maintanence := FALSE;
   STATUS[863].EXT.Operation := FALSE;
   STATUS[863].EXT.Forced := FALSE;
   STATUS[863].EXT.BIT29 := FALSE;
   STATUS[863].EXT.BIT30 := FALSE;
   STATUS[863].EXT.BIT31 := FALSE;
   STATUS[863].EXT.ModeBit1 := FALSE;
   STATUS[863].EXT.ModeBit2 := FALSE;
   STATUS[863].EXT.ModeBit3 := FALSE;
   STATUS[863].EXT.BIT19 := FALSE;
   STATUS[863].EXT.BIT20 := FALSE;
   STATUS[863].EXT.AlarmSuppressed := FALSE;
   STATUS[863].EXT.AlarmPrsent := FALSE;
   STATUS[863].EXT.AlarmFailUnAck := FALSE;
   STATUS[863].Status := 0;
   STATUS[863].TimeStamp := 16#0000;
   STATUS[864].VALUE := 0.0;
   STATUS[864].TRIGVALUE := 0.0;
   STATUS[864].EXT.AlarmWarnUnAck := FALSE;
   STATUS[864].EXT.AckRequired := FALSE;
   STATUS[864].EXT.Maintanence := FALSE;
   STATUS[864].EXT.Operation := FALSE;
   STATUS[864].EXT.Forced := FALSE;
   STATUS[864].EXT.BIT29 := FALSE;
   STATUS[864].EXT.BIT30 := FALSE;
   STATUS[864].EXT.BIT31 := FALSE;
   STATUS[864].EXT.ModeBit1 := FALSE;
   STATUS[864].EXT.ModeBit2 := FALSE;
   STATUS[864].EXT.ModeBit3 := FALSE;
   STATUS[864].EXT.BIT19 := FALSE;
   STATUS[864].EXT.BIT20 := FALSE;
   STATUS[864].EXT.AlarmSuppressed := FALSE;
   STATUS[864].EXT.AlarmPrsent := FALSE;
   STATUS[864].EXT.AlarmFailUnAck := FALSE;
   STATUS[864].Status := 0;
   STATUS[864].TimeStamp := 16#0000;
   STATUS[865].VALUE := 0.0;
   STATUS[865].TRIGVALUE := 0.0;
   STATUS[865].EXT.AlarmWarnUnAck := FALSE;
   STATUS[865].EXT.AckRequired := FALSE;
   STATUS[865].EXT.Maintanence := FALSE;
   STATUS[865].EXT.Operation := FALSE;
   STATUS[865].EXT.Forced := FALSE;
   STATUS[865].EXT.BIT29 := FALSE;
   STATUS[865].EXT.BIT30 := FALSE;
   STATUS[865].EXT.BIT31 := FALSE;
   STATUS[865].EXT.ModeBit1 := FALSE;
   STATUS[865].EXT.ModeBit2 := FALSE;
   STATUS[865].EXT.ModeBit3 := FALSE;
   STATUS[865].EXT.BIT19 := FALSE;
   STATUS[865].EXT.BIT20 := FALSE;
   STATUS[865].EXT.AlarmSuppressed := FALSE;
   STATUS[865].EXT.AlarmPrsent := FALSE;
   STATUS[865].EXT.AlarmFailUnAck := FALSE;
   STATUS[865].Status := 0;
   STATUS[865].TimeStamp := 16#0000;
   STATUS[866].VALUE := 0.0;
   STATUS[866].TRIGVALUE := 0.0;
   STATUS[866].EXT.AlarmWarnUnAck := FALSE;
   STATUS[866].EXT.AckRequired := FALSE;
   STATUS[866].EXT.Maintanence := FALSE;
   STATUS[866].EXT.Operation := FALSE;
   STATUS[866].EXT.Forced := FALSE;
   STATUS[866].EXT.BIT29 := FALSE;
   STATUS[866].EXT.BIT30 := FALSE;
   STATUS[866].EXT.BIT31 := FALSE;
   STATUS[866].EXT.ModeBit1 := FALSE;
   STATUS[866].EXT.ModeBit2 := FALSE;
   STATUS[866].EXT.ModeBit3 := FALSE;
   STATUS[866].EXT.BIT19 := FALSE;
   STATUS[866].EXT.BIT20 := FALSE;
   STATUS[866].EXT.AlarmSuppressed := FALSE;
   STATUS[866].EXT.AlarmPrsent := FALSE;
   STATUS[866].EXT.AlarmFailUnAck := FALSE;
   STATUS[866].Status := 0;
   STATUS[866].TimeStamp := 16#0000;
   STATUS[867].VALUE := 0.0;
   STATUS[867].TRIGVALUE := 0.0;
   STATUS[867].EXT.AlarmWarnUnAck := FALSE;
   STATUS[867].EXT.AckRequired := FALSE;
   STATUS[867].EXT.Maintanence := FALSE;
   STATUS[867].EXT.Operation := FALSE;
   STATUS[867].EXT.Forced := FALSE;
   STATUS[867].EXT.BIT29 := FALSE;
   STATUS[867].EXT.BIT30 := FALSE;
   STATUS[867].EXT.BIT31 := FALSE;
   STATUS[867].EXT.ModeBit1 := FALSE;
   STATUS[867].EXT.ModeBit2 := FALSE;
   STATUS[867].EXT.ModeBit3 := FALSE;
   STATUS[867].EXT.BIT19 := FALSE;
   STATUS[867].EXT.BIT20 := FALSE;
   STATUS[867].EXT.AlarmSuppressed := FALSE;
   STATUS[867].EXT.AlarmPrsent := FALSE;
   STATUS[867].EXT.AlarmFailUnAck := FALSE;
   STATUS[867].Status := 0;
   STATUS[867].TimeStamp := 16#0000;
   STATUS[868].VALUE := 0.0;
   STATUS[868].TRIGVALUE := 0.0;
   STATUS[868].EXT.AlarmWarnUnAck := FALSE;
   STATUS[868].EXT.AckRequired := FALSE;
   STATUS[868].EXT.Maintanence := FALSE;
   STATUS[868].EXT.Operation := FALSE;
   STATUS[868].EXT.Forced := FALSE;
   STATUS[868].EXT.BIT29 := FALSE;
   STATUS[868].EXT.BIT30 := FALSE;
   STATUS[868].EXT.BIT31 := FALSE;
   STATUS[868].EXT.ModeBit1 := FALSE;
   STATUS[868].EXT.ModeBit2 := FALSE;
   STATUS[868].EXT.ModeBit3 := FALSE;
   STATUS[868].EXT.BIT19 := FALSE;
   STATUS[868].EXT.BIT20 := FALSE;
   STATUS[868].EXT.AlarmSuppressed := FALSE;
   STATUS[868].EXT.AlarmPrsent := FALSE;
   STATUS[868].EXT.AlarmFailUnAck := FALSE;
   STATUS[868].Status := 0;
   STATUS[868].TimeStamp := 16#0000;
   STATUS[869].VALUE := 0.0;
   STATUS[869].TRIGVALUE := 0.0;
   STATUS[869].EXT.AlarmWarnUnAck := FALSE;
   STATUS[869].EXT.AckRequired := FALSE;
   STATUS[869].EXT.Maintanence := FALSE;
   STATUS[869].EXT.Operation := FALSE;
   STATUS[869].EXT.Forced := FALSE;
   STATUS[869].EXT.BIT29 := FALSE;
   STATUS[869].EXT.BIT30 := FALSE;
   STATUS[869].EXT.BIT31 := FALSE;
   STATUS[869].EXT.ModeBit1 := FALSE;
   STATUS[869].EXT.ModeBit2 := FALSE;
   STATUS[869].EXT.ModeBit3 := FALSE;
   STATUS[869].EXT.BIT19 := FALSE;
   STATUS[869].EXT.BIT20 := FALSE;
   STATUS[869].EXT.AlarmSuppressed := FALSE;
   STATUS[869].EXT.AlarmPrsent := FALSE;
   STATUS[869].EXT.AlarmFailUnAck := FALSE;
   STATUS[869].Status := 0;
   STATUS[869].TimeStamp := 16#0000;
   STATUS[870].VALUE := 0.0;
   STATUS[870].TRIGVALUE := 0.0;
   STATUS[870].EXT.AlarmWarnUnAck := FALSE;
   STATUS[870].EXT.AckRequired := FALSE;
   STATUS[870].EXT.Maintanence := FALSE;
   STATUS[870].EXT.Operation := FALSE;
   STATUS[870].EXT.Forced := FALSE;
   STATUS[870].EXT.BIT29 := FALSE;
   STATUS[870].EXT.BIT30 := FALSE;
   STATUS[870].EXT.BIT31 := FALSE;
   STATUS[870].EXT.ModeBit1 := FALSE;
   STATUS[870].EXT.ModeBit2 := FALSE;
   STATUS[870].EXT.ModeBit3 := FALSE;
   STATUS[870].EXT.BIT19 := FALSE;
   STATUS[870].EXT.BIT20 := FALSE;
   STATUS[870].EXT.AlarmSuppressed := FALSE;
   STATUS[870].EXT.AlarmPrsent := FALSE;
   STATUS[870].EXT.AlarmFailUnAck := FALSE;
   STATUS[870].Status := 0;
   STATUS[870].TimeStamp := 16#0000;
   STATUS[871].VALUE := 0.0;
   STATUS[871].TRIGVALUE := 0.0;
   STATUS[871].EXT.AlarmWarnUnAck := FALSE;
   STATUS[871].EXT.AckRequired := FALSE;
   STATUS[871].EXT.Maintanence := FALSE;
   STATUS[871].EXT.Operation := FALSE;
   STATUS[871].EXT.Forced := FALSE;
   STATUS[871].EXT.BIT29 := FALSE;
   STATUS[871].EXT.BIT30 := FALSE;
   STATUS[871].EXT.BIT31 := FALSE;
   STATUS[871].EXT.ModeBit1 := FALSE;
   STATUS[871].EXT.ModeBit2 := FALSE;
   STATUS[871].EXT.ModeBit3 := FALSE;
   STATUS[871].EXT.BIT19 := FALSE;
   STATUS[871].EXT.BIT20 := FALSE;
   STATUS[871].EXT.AlarmSuppressed := FALSE;
   STATUS[871].EXT.AlarmPrsent := FALSE;
   STATUS[871].EXT.AlarmFailUnAck := FALSE;
   STATUS[871].Status := 0;
   STATUS[871].TimeStamp := 16#0000;
   STATUS[872].VALUE := 0.0;
   STATUS[872].TRIGVALUE := 0.0;
   STATUS[872].EXT.AlarmWarnUnAck := FALSE;
   STATUS[872].EXT.AckRequired := FALSE;
   STATUS[872].EXT.Maintanence := FALSE;
   STATUS[872].EXT.Operation := FALSE;
   STATUS[872].EXT.Forced := FALSE;
   STATUS[872].EXT.BIT29 := FALSE;
   STATUS[872].EXT.BIT30 := FALSE;
   STATUS[872].EXT.BIT31 := FALSE;
   STATUS[872].EXT.ModeBit1 := FALSE;
   STATUS[872].EXT.ModeBit2 := FALSE;
   STATUS[872].EXT.ModeBit3 := FALSE;
   STATUS[872].EXT.BIT19 := FALSE;
   STATUS[872].EXT.BIT20 := FALSE;
   STATUS[872].EXT.AlarmSuppressed := FALSE;
   STATUS[872].EXT.AlarmPrsent := FALSE;
   STATUS[872].EXT.AlarmFailUnAck := FALSE;
   STATUS[872].Status := 0;
   STATUS[872].TimeStamp := 16#0000;
   STATUS[873].VALUE := 0.0;
   STATUS[873].TRIGVALUE := 0.0;
   STATUS[873].EXT.AlarmWarnUnAck := FALSE;
   STATUS[873].EXT.AckRequired := FALSE;
   STATUS[873].EXT.Maintanence := FALSE;
   STATUS[873].EXT.Operation := FALSE;
   STATUS[873].EXT.Forced := FALSE;
   STATUS[873].EXT.BIT29 := FALSE;
   STATUS[873].EXT.BIT30 := FALSE;
   STATUS[873].EXT.BIT31 := FALSE;
   STATUS[873].EXT.ModeBit1 := FALSE;
   STATUS[873].EXT.ModeBit2 := FALSE;
   STATUS[873].EXT.ModeBit3 := FALSE;
   STATUS[873].EXT.BIT19 := FALSE;
   STATUS[873].EXT.BIT20 := FALSE;
   STATUS[873].EXT.AlarmSuppressed := FALSE;
   STATUS[873].EXT.AlarmPrsent := FALSE;
   STATUS[873].EXT.AlarmFailUnAck := FALSE;
   STATUS[873].Status := 0;
   STATUS[873].TimeStamp := 16#0000;
   STATUS[874].VALUE := 0.0;
   STATUS[874].TRIGVALUE := 0.0;
   STATUS[874].EXT.AlarmWarnUnAck := FALSE;
   STATUS[874].EXT.AckRequired := FALSE;
   STATUS[874].EXT.Maintanence := FALSE;
   STATUS[874].EXT.Operation := FALSE;
   STATUS[874].EXT.Forced := FALSE;
   STATUS[874].EXT.BIT29 := FALSE;
   STATUS[874].EXT.BIT30 := FALSE;
   STATUS[874].EXT.BIT31 := FALSE;
   STATUS[874].EXT.ModeBit1 := FALSE;
   STATUS[874].EXT.ModeBit2 := FALSE;
   STATUS[874].EXT.ModeBit3 := FALSE;
   STATUS[874].EXT.BIT19 := FALSE;
   STATUS[874].EXT.BIT20 := FALSE;
   STATUS[874].EXT.AlarmSuppressed := FALSE;
   STATUS[874].EXT.AlarmPrsent := FALSE;
   STATUS[874].EXT.AlarmFailUnAck := FALSE;
   STATUS[874].Status := 0;
   STATUS[874].TimeStamp := 16#0000;
   STATUS[875].VALUE := 0.0;
   STATUS[875].TRIGVALUE := 0.0;
   STATUS[875].EXT.AlarmWarnUnAck := FALSE;
   STATUS[875].EXT.AckRequired := FALSE;
   STATUS[875].EXT.Maintanence := FALSE;
   STATUS[875].EXT.Operation := FALSE;
   STATUS[875].EXT.Forced := FALSE;
   STATUS[875].EXT.BIT29 := FALSE;
   STATUS[875].EXT.BIT30 := FALSE;
   STATUS[875].EXT.BIT31 := FALSE;
   STATUS[875].EXT.ModeBit1 := FALSE;
   STATUS[875].EXT.ModeBit2 := FALSE;
   STATUS[875].EXT.ModeBit3 := FALSE;
   STATUS[875].EXT.BIT19 := FALSE;
   STATUS[875].EXT.BIT20 := FALSE;
   STATUS[875].EXT.AlarmSuppressed := FALSE;
   STATUS[875].EXT.AlarmPrsent := FALSE;
   STATUS[875].EXT.AlarmFailUnAck := FALSE;
   STATUS[875].Status := 0;
   STATUS[875].TimeStamp := 16#0000;
   STATUS[876].VALUE := 0.0;
   STATUS[876].TRIGVALUE := 0.0;
   STATUS[876].EXT.AlarmWarnUnAck := FALSE;
   STATUS[876].EXT.AckRequired := FALSE;
   STATUS[876].EXT.Maintanence := FALSE;
   STATUS[876].EXT.Operation := FALSE;
   STATUS[876].EXT.Forced := FALSE;
   STATUS[876].EXT.BIT29 := FALSE;
   STATUS[876].EXT.BIT30 := FALSE;
   STATUS[876].EXT.BIT31 := FALSE;
   STATUS[876].EXT.ModeBit1 := FALSE;
   STATUS[876].EXT.ModeBit2 := FALSE;
   STATUS[876].EXT.ModeBit3 := FALSE;
   STATUS[876].EXT.BIT19 := FALSE;
   STATUS[876].EXT.BIT20 := FALSE;
   STATUS[876].EXT.AlarmSuppressed := FALSE;
   STATUS[876].EXT.AlarmPrsent := FALSE;
   STATUS[876].EXT.AlarmFailUnAck := FALSE;
   STATUS[876].Status := 0;
   STATUS[876].TimeStamp := 16#0000;
   STATUS[877].VALUE := 0.0;
   STATUS[877].TRIGVALUE := 0.0;
   STATUS[877].EXT.AlarmWarnUnAck := FALSE;
   STATUS[877].EXT.AckRequired := FALSE;
   STATUS[877].EXT.Maintanence := FALSE;
   STATUS[877].EXT.Operation := FALSE;
   STATUS[877].EXT.Forced := FALSE;
   STATUS[877].EXT.BIT29 := FALSE;
   STATUS[877].EXT.BIT30 := FALSE;
   STATUS[877].EXT.BIT31 := FALSE;
   STATUS[877].EXT.ModeBit1 := FALSE;
   STATUS[877].EXT.ModeBit2 := FALSE;
   STATUS[877].EXT.ModeBit3 := FALSE;
   STATUS[877].EXT.BIT19 := FALSE;
   STATUS[877].EXT.BIT20 := FALSE;
   STATUS[877].EXT.AlarmSuppressed := FALSE;
   STATUS[877].EXT.AlarmPrsent := FALSE;
   STATUS[877].EXT.AlarmFailUnAck := FALSE;
   STATUS[877].Status := 0;
   STATUS[877].TimeStamp := 16#0000;
   STATUS[878].VALUE := 0.0;
   STATUS[878].TRIGVALUE := 0.0;
   STATUS[878].EXT.AlarmWarnUnAck := FALSE;
   STATUS[878].EXT.AckRequired := FALSE;
   STATUS[878].EXT.Maintanence := FALSE;
   STATUS[878].EXT.Operation := FALSE;
   STATUS[878].EXT.Forced := FALSE;
   STATUS[878].EXT.BIT29 := FALSE;
   STATUS[878].EXT.BIT30 := FALSE;
   STATUS[878].EXT.BIT31 := FALSE;
   STATUS[878].EXT.ModeBit1 := FALSE;
   STATUS[878].EXT.ModeBit2 := FALSE;
   STATUS[878].EXT.ModeBit3 := FALSE;
   STATUS[878].EXT.BIT19 := FALSE;
   STATUS[878].EXT.BIT20 := FALSE;
   STATUS[878].EXT.AlarmSuppressed := FALSE;
   STATUS[878].EXT.AlarmPrsent := FALSE;
   STATUS[878].EXT.AlarmFailUnAck := FALSE;
   STATUS[878].Status := 0;
   STATUS[878].TimeStamp := 16#0000;
   STATUS[879].VALUE := 0.0;
   STATUS[879].TRIGVALUE := 0.0;
   STATUS[879].EXT.AlarmWarnUnAck := FALSE;
   STATUS[879].EXT.AckRequired := FALSE;
   STATUS[879].EXT.Maintanence := FALSE;
   STATUS[879].EXT.Operation := FALSE;
   STATUS[879].EXT.Forced := FALSE;
   STATUS[879].EXT.BIT29 := FALSE;
   STATUS[879].EXT.BIT30 := FALSE;
   STATUS[879].EXT.BIT31 := FALSE;
   STATUS[879].EXT.ModeBit1 := FALSE;
   STATUS[879].EXT.ModeBit2 := FALSE;
   STATUS[879].EXT.ModeBit3 := FALSE;
   STATUS[879].EXT.BIT19 := FALSE;
   STATUS[879].EXT.BIT20 := FALSE;
   STATUS[879].EXT.AlarmSuppressed := FALSE;
   STATUS[879].EXT.AlarmPrsent := FALSE;
   STATUS[879].EXT.AlarmFailUnAck := FALSE;
   STATUS[879].Status := 0;
   STATUS[879].TimeStamp := 16#0000;
   STATUS[880].VALUE := 0.0;
   STATUS[880].TRIGVALUE := 0.0;
   STATUS[880].EXT.AlarmWarnUnAck := FALSE;
   STATUS[880].EXT.AckRequired := FALSE;
   STATUS[880].EXT.Maintanence := FALSE;
   STATUS[880].EXT.Operation := FALSE;
   STATUS[880].EXT.Forced := FALSE;
   STATUS[880].EXT.BIT29 := FALSE;
   STATUS[880].EXT.BIT30 := FALSE;
   STATUS[880].EXT.BIT31 := FALSE;
   STATUS[880].EXT.ModeBit1 := FALSE;
   STATUS[880].EXT.ModeBit2 := FALSE;
   STATUS[880].EXT.ModeBit3 := FALSE;
   STATUS[880].EXT.BIT19 := FALSE;
   STATUS[880].EXT.BIT20 := FALSE;
   STATUS[880].EXT.AlarmSuppressed := FALSE;
   STATUS[880].EXT.AlarmPrsent := FALSE;
   STATUS[880].EXT.AlarmFailUnAck := FALSE;
   STATUS[880].Status := 0;
   STATUS[880].TimeStamp := 16#0000;
   STATUS[881].VALUE := 0.0;
   STATUS[881].TRIGVALUE := 0.0;
   STATUS[881].EXT.AlarmWarnUnAck := FALSE;
   STATUS[881].EXT.AckRequired := FALSE;
   STATUS[881].EXT.Maintanence := FALSE;
   STATUS[881].EXT.Operation := FALSE;
   STATUS[881].EXT.Forced := FALSE;
   STATUS[881].EXT.BIT29 := FALSE;
   STATUS[881].EXT.BIT30 := FALSE;
   STATUS[881].EXT.BIT31 := FALSE;
   STATUS[881].EXT.ModeBit1 := FALSE;
   STATUS[881].EXT.ModeBit2 := FALSE;
   STATUS[881].EXT.ModeBit3 := FALSE;
   STATUS[881].EXT.BIT19 := FALSE;
   STATUS[881].EXT.BIT20 := FALSE;
   STATUS[881].EXT.AlarmSuppressed := FALSE;
   STATUS[881].EXT.AlarmPrsent := FALSE;
   STATUS[881].EXT.AlarmFailUnAck := FALSE;
   STATUS[881].Status := 0;
   STATUS[881].TimeStamp := 16#0000;
   STATUS[882].VALUE := 0.0;
   STATUS[882].TRIGVALUE := 0.0;
   STATUS[882].EXT.AlarmWarnUnAck := FALSE;
   STATUS[882].EXT.AckRequired := FALSE;
   STATUS[882].EXT.Maintanence := FALSE;
   STATUS[882].EXT.Operation := FALSE;
   STATUS[882].EXT.Forced := FALSE;
   STATUS[882].EXT.BIT29 := FALSE;
   STATUS[882].EXT.BIT30 := FALSE;
   STATUS[882].EXT.BIT31 := FALSE;
   STATUS[882].EXT.ModeBit1 := FALSE;
   STATUS[882].EXT.ModeBit2 := FALSE;
   STATUS[882].EXT.ModeBit3 := FALSE;
   STATUS[882].EXT.BIT19 := FALSE;
   STATUS[882].EXT.BIT20 := FALSE;
   STATUS[882].EXT.AlarmSuppressed := FALSE;
   STATUS[882].EXT.AlarmPrsent := FALSE;
   STATUS[882].EXT.AlarmFailUnAck := FALSE;
   STATUS[882].Status := 0;
   STATUS[882].TimeStamp := 16#0000;
   STATUS[883].VALUE := 0.0;
   STATUS[883].TRIGVALUE := 0.0;
   STATUS[883].EXT.AlarmWarnUnAck := FALSE;
   STATUS[883].EXT.AckRequired := FALSE;
   STATUS[883].EXT.Maintanence := FALSE;
   STATUS[883].EXT.Operation := FALSE;
   STATUS[883].EXT.Forced := FALSE;
   STATUS[883].EXT.BIT29 := FALSE;
   STATUS[883].EXT.BIT30 := FALSE;
   STATUS[883].EXT.BIT31 := FALSE;
   STATUS[883].EXT.ModeBit1 := FALSE;
   STATUS[883].EXT.ModeBit2 := FALSE;
   STATUS[883].EXT.ModeBit3 := FALSE;
   STATUS[883].EXT.BIT19 := FALSE;
   STATUS[883].EXT.BIT20 := FALSE;
   STATUS[883].EXT.AlarmSuppressed := FALSE;
   STATUS[883].EXT.AlarmPrsent := FALSE;
   STATUS[883].EXT.AlarmFailUnAck := FALSE;
   STATUS[883].Status := 0;
   STATUS[883].TimeStamp := 16#0000;
   STATUS[884].VALUE := 0.0;
   STATUS[884].TRIGVALUE := 0.0;
   STATUS[884].EXT.AlarmWarnUnAck := FALSE;
   STATUS[884].EXT.AckRequired := FALSE;
   STATUS[884].EXT.Maintanence := FALSE;
   STATUS[884].EXT.Operation := FALSE;
   STATUS[884].EXT.Forced := FALSE;
   STATUS[884].EXT.BIT29 := FALSE;
   STATUS[884].EXT.BIT30 := FALSE;
   STATUS[884].EXT.BIT31 := FALSE;
   STATUS[884].EXT.ModeBit1 := FALSE;
   STATUS[884].EXT.ModeBit2 := FALSE;
   STATUS[884].EXT.ModeBit3 := FALSE;
   STATUS[884].EXT.BIT19 := FALSE;
   STATUS[884].EXT.BIT20 := FALSE;
   STATUS[884].EXT.AlarmSuppressed := FALSE;
   STATUS[884].EXT.AlarmPrsent := FALSE;
   STATUS[884].EXT.AlarmFailUnAck := FALSE;
   STATUS[884].Status := 0;
   STATUS[884].TimeStamp := 16#0000;
   STATUS[885].VALUE := 0.0;
   STATUS[885].TRIGVALUE := 0.0;
   STATUS[885].EXT.AlarmWarnUnAck := FALSE;
   STATUS[885].EXT.AckRequired := FALSE;
   STATUS[885].EXT.Maintanence := FALSE;
   STATUS[885].EXT.Operation := FALSE;
   STATUS[885].EXT.Forced := FALSE;
   STATUS[885].EXT.BIT29 := FALSE;
   STATUS[885].EXT.BIT30 := FALSE;
   STATUS[885].EXT.BIT31 := FALSE;
   STATUS[885].EXT.ModeBit1 := FALSE;
   STATUS[885].EXT.ModeBit2 := FALSE;
   STATUS[885].EXT.ModeBit3 := FALSE;
   STATUS[885].EXT.BIT19 := FALSE;
   STATUS[885].EXT.BIT20 := FALSE;
   STATUS[885].EXT.AlarmSuppressed := FALSE;
   STATUS[885].EXT.AlarmPrsent := FALSE;
   STATUS[885].EXT.AlarmFailUnAck := FALSE;
   STATUS[885].Status := 0;
   STATUS[885].TimeStamp := 16#0000;
   STATUS[886].VALUE := 0.0;
   STATUS[886].TRIGVALUE := 0.0;
   STATUS[886].EXT.AlarmWarnUnAck := FALSE;
   STATUS[886].EXT.AckRequired := FALSE;
   STATUS[886].EXT.Maintanence := FALSE;
   STATUS[886].EXT.Operation := FALSE;
   STATUS[886].EXT.Forced := FALSE;
   STATUS[886].EXT.BIT29 := FALSE;
   STATUS[886].EXT.BIT30 := FALSE;
   STATUS[886].EXT.BIT31 := FALSE;
   STATUS[886].EXT.ModeBit1 := FALSE;
   STATUS[886].EXT.ModeBit2 := FALSE;
   STATUS[886].EXT.ModeBit3 := FALSE;
   STATUS[886].EXT.BIT19 := FALSE;
   STATUS[886].EXT.BIT20 := FALSE;
   STATUS[886].EXT.AlarmSuppressed := FALSE;
   STATUS[886].EXT.AlarmPrsent := FALSE;
   STATUS[886].EXT.AlarmFailUnAck := FALSE;
   STATUS[886].Status := 0;
   STATUS[886].TimeStamp := 16#0000;
   STATUS[887].VALUE := 0.0;
   STATUS[887].TRIGVALUE := 0.0;
   STATUS[887].EXT.AlarmWarnUnAck := FALSE;
   STATUS[887].EXT.AckRequired := FALSE;
   STATUS[887].EXT.Maintanence := FALSE;
   STATUS[887].EXT.Operation := FALSE;
   STATUS[887].EXT.Forced := FALSE;
   STATUS[887].EXT.BIT29 := FALSE;
   STATUS[887].EXT.BIT30 := FALSE;
   STATUS[887].EXT.BIT31 := FALSE;
   STATUS[887].EXT.ModeBit1 := FALSE;
   STATUS[887].EXT.ModeBit2 := FALSE;
   STATUS[887].EXT.ModeBit3 := FALSE;
   STATUS[887].EXT.BIT19 := FALSE;
   STATUS[887].EXT.BIT20 := FALSE;
   STATUS[887].EXT.AlarmSuppressed := FALSE;
   STATUS[887].EXT.AlarmPrsent := FALSE;
   STATUS[887].EXT.AlarmFailUnAck := FALSE;
   STATUS[887].Status := 0;
   STATUS[887].TimeStamp := 16#0000;
   STATUS[888].VALUE := 0.0;
   STATUS[888].TRIGVALUE := 0.0;
   STATUS[888].EXT.AlarmWarnUnAck := FALSE;
   STATUS[888].EXT.AckRequired := FALSE;
   STATUS[888].EXT.Maintanence := FALSE;
   STATUS[888].EXT.Operation := FALSE;
   STATUS[888].EXT.Forced := FALSE;
   STATUS[888].EXT.BIT29 := FALSE;
   STATUS[888].EXT.BIT30 := FALSE;
   STATUS[888].EXT.BIT31 := FALSE;
   STATUS[888].EXT.ModeBit1 := FALSE;
   STATUS[888].EXT.ModeBit2 := FALSE;
   STATUS[888].EXT.ModeBit3 := FALSE;
   STATUS[888].EXT.BIT19 := FALSE;
   STATUS[888].EXT.BIT20 := FALSE;
   STATUS[888].EXT.AlarmSuppressed := FALSE;
   STATUS[888].EXT.AlarmPrsent := FALSE;
   STATUS[888].EXT.AlarmFailUnAck := FALSE;
   STATUS[888].Status := 0;
   STATUS[888].TimeStamp := 16#0000;
   STATUS[889].VALUE := 0.0;
   STATUS[889].TRIGVALUE := 0.0;
   STATUS[889].EXT.AlarmWarnUnAck := FALSE;
   STATUS[889].EXT.AckRequired := FALSE;
   STATUS[889].EXT.Maintanence := FALSE;
   STATUS[889].EXT.Operation := FALSE;
   STATUS[889].EXT.Forced := FALSE;
   STATUS[889].EXT.BIT29 := FALSE;
   STATUS[889].EXT.BIT30 := FALSE;
   STATUS[889].EXT.BIT31 := FALSE;
   STATUS[889].EXT.ModeBit1 := FALSE;
   STATUS[889].EXT.ModeBit2 := FALSE;
   STATUS[889].EXT.ModeBit3 := FALSE;
   STATUS[889].EXT.BIT19 := FALSE;
   STATUS[889].EXT.BIT20 := FALSE;
   STATUS[889].EXT.AlarmSuppressed := FALSE;
   STATUS[889].EXT.AlarmPrsent := FALSE;
   STATUS[889].EXT.AlarmFailUnAck := FALSE;
   STATUS[889].Status := 0;
   STATUS[889].TimeStamp := 16#0000;
   STATUS[890].VALUE := 0.0;
   STATUS[890].TRIGVALUE := 0.0;
   STATUS[890].EXT.AlarmWarnUnAck := FALSE;
   STATUS[890].EXT.AckRequired := FALSE;
   STATUS[890].EXT.Maintanence := FALSE;
   STATUS[890].EXT.Operation := FALSE;
   STATUS[890].EXT.Forced := FALSE;
   STATUS[890].EXT.BIT29 := FALSE;
   STATUS[890].EXT.BIT30 := FALSE;
   STATUS[890].EXT.BIT31 := FALSE;
   STATUS[890].EXT.ModeBit1 := FALSE;
   STATUS[890].EXT.ModeBit2 := FALSE;
   STATUS[890].EXT.ModeBit3 := FALSE;
   STATUS[890].EXT.BIT19 := FALSE;
   STATUS[890].EXT.BIT20 := FALSE;
   STATUS[890].EXT.AlarmSuppressed := FALSE;
   STATUS[890].EXT.AlarmPrsent := FALSE;
   STATUS[890].EXT.AlarmFailUnAck := FALSE;
   STATUS[890].Status := 0;
   STATUS[890].TimeStamp := 16#0000;
   STATUS[891].VALUE := 0.0;
   STATUS[891].TRIGVALUE := 0.0;
   STATUS[891].EXT.AlarmWarnUnAck := FALSE;
   STATUS[891].EXT.AckRequired := FALSE;
   STATUS[891].EXT.Maintanence := FALSE;
   STATUS[891].EXT.Operation := FALSE;
   STATUS[891].EXT.Forced := FALSE;
   STATUS[891].EXT.BIT29 := FALSE;
   STATUS[891].EXT.BIT30 := FALSE;
   STATUS[891].EXT.BIT31 := FALSE;
   STATUS[891].EXT.ModeBit1 := FALSE;
   STATUS[891].EXT.ModeBit2 := FALSE;
   STATUS[891].EXT.ModeBit3 := FALSE;
   STATUS[891].EXT.BIT19 := FALSE;
   STATUS[891].EXT.BIT20 := FALSE;
   STATUS[891].EXT.AlarmSuppressed := FALSE;
   STATUS[891].EXT.AlarmPrsent := FALSE;
   STATUS[891].EXT.AlarmFailUnAck := FALSE;
   STATUS[891].Status := 0;
   STATUS[891].TimeStamp := 16#0000;
   STATUS[892].VALUE := 0.0;
   STATUS[892].TRIGVALUE := 0.0;
   STATUS[892].EXT.AlarmWarnUnAck := FALSE;
   STATUS[892].EXT.AckRequired := FALSE;
   STATUS[892].EXT.Maintanence := FALSE;
   STATUS[892].EXT.Operation := FALSE;
   STATUS[892].EXT.Forced := FALSE;
   STATUS[892].EXT.BIT29 := FALSE;
   STATUS[892].EXT.BIT30 := FALSE;
   STATUS[892].EXT.BIT31 := FALSE;
   STATUS[892].EXT.ModeBit1 := FALSE;
   STATUS[892].EXT.ModeBit2 := FALSE;
   STATUS[892].EXT.ModeBit3 := FALSE;
   STATUS[892].EXT.BIT19 := FALSE;
   STATUS[892].EXT.BIT20 := FALSE;
   STATUS[892].EXT.AlarmSuppressed := FALSE;
   STATUS[892].EXT.AlarmPrsent := FALSE;
   STATUS[892].EXT.AlarmFailUnAck := FALSE;
   STATUS[892].Status := 0;
   STATUS[892].TimeStamp := 16#0000;
   STATUS[893].VALUE := 0.0;
   STATUS[893].TRIGVALUE := 0.0;
   STATUS[893].EXT.AlarmWarnUnAck := FALSE;
   STATUS[893].EXT.AckRequired := FALSE;
   STATUS[893].EXT.Maintanence := FALSE;
   STATUS[893].EXT.Operation := FALSE;
   STATUS[893].EXT.Forced := FALSE;
   STATUS[893].EXT.BIT29 := FALSE;
   STATUS[893].EXT.BIT30 := FALSE;
   STATUS[893].EXT.BIT31 := FALSE;
   STATUS[893].EXT.ModeBit1 := FALSE;
   STATUS[893].EXT.ModeBit2 := FALSE;
   STATUS[893].EXT.ModeBit3 := FALSE;
   STATUS[893].EXT.BIT19 := FALSE;
   STATUS[893].EXT.BIT20 := FALSE;
   STATUS[893].EXT.AlarmSuppressed := FALSE;
   STATUS[893].EXT.AlarmPrsent := FALSE;
   STATUS[893].EXT.AlarmFailUnAck := FALSE;
   STATUS[893].Status := 0;
   STATUS[893].TimeStamp := 16#0000;
   STATUS[894].VALUE := 0.0;
   STATUS[894].TRIGVALUE := 0.0;
   STATUS[894].EXT.AlarmWarnUnAck := FALSE;
   STATUS[894].EXT.AckRequired := FALSE;
   STATUS[894].EXT.Maintanence := FALSE;
   STATUS[894].EXT.Operation := FALSE;
   STATUS[894].EXT.Forced := FALSE;
   STATUS[894].EXT.BIT29 := FALSE;
   STATUS[894].EXT.BIT30 := FALSE;
   STATUS[894].EXT.BIT31 := FALSE;
   STATUS[894].EXT.ModeBit1 := FALSE;
   STATUS[894].EXT.ModeBit2 := FALSE;
   STATUS[894].EXT.ModeBit3 := FALSE;
   STATUS[894].EXT.BIT19 := FALSE;
   STATUS[894].EXT.BIT20 := FALSE;
   STATUS[894].EXT.AlarmSuppressed := FALSE;
   STATUS[894].EXT.AlarmPrsent := FALSE;
   STATUS[894].EXT.AlarmFailUnAck := FALSE;
   STATUS[894].Status := 0;
   STATUS[894].TimeStamp := 16#0000;
   STATUS[895].VALUE := 0.0;
   STATUS[895].TRIGVALUE := 0.0;
   STATUS[895].EXT.AlarmWarnUnAck := FALSE;
   STATUS[895].EXT.AckRequired := FALSE;
   STATUS[895].EXT.Maintanence := FALSE;
   STATUS[895].EXT.Operation := FALSE;
   STATUS[895].EXT.Forced := FALSE;
   STATUS[895].EXT.BIT29 := FALSE;
   STATUS[895].EXT.BIT30 := FALSE;
   STATUS[895].EXT.BIT31 := FALSE;
   STATUS[895].EXT.ModeBit1 := FALSE;
   STATUS[895].EXT.ModeBit2 := FALSE;
   STATUS[895].EXT.ModeBit3 := FALSE;
   STATUS[895].EXT.BIT19 := FALSE;
   STATUS[895].EXT.BIT20 := FALSE;
   STATUS[895].EXT.AlarmSuppressed := FALSE;
   STATUS[895].EXT.AlarmPrsent := FALSE;
   STATUS[895].EXT.AlarmFailUnAck := FALSE;
   STATUS[895].Status := 0;
   STATUS[895].TimeStamp := 16#0000;
   STATUS[896].VALUE := 0.0;
   STATUS[896].TRIGVALUE := 0.0;
   STATUS[896].EXT.AlarmWarnUnAck := FALSE;
   STATUS[896].EXT.AckRequired := FALSE;
   STATUS[896].EXT.Maintanence := FALSE;
   STATUS[896].EXT.Operation := FALSE;
   STATUS[896].EXT.Forced := FALSE;
   STATUS[896].EXT.BIT29 := FALSE;
   STATUS[896].EXT.BIT30 := FALSE;
   STATUS[896].EXT.BIT31 := FALSE;
   STATUS[896].EXT.ModeBit1 := FALSE;
   STATUS[896].EXT.ModeBit2 := FALSE;
   STATUS[896].EXT.ModeBit3 := FALSE;
   STATUS[896].EXT.BIT19 := FALSE;
   STATUS[896].EXT.BIT20 := FALSE;
   STATUS[896].EXT.AlarmSuppressed := FALSE;
   STATUS[896].EXT.AlarmPrsent := FALSE;
   STATUS[896].EXT.AlarmFailUnAck := FALSE;
   STATUS[896].Status := 0;
   STATUS[896].TimeStamp := 16#0000;
   STATUS[897].VALUE := 0.0;
   STATUS[897].TRIGVALUE := 0.0;
   STATUS[897].EXT.AlarmWarnUnAck := FALSE;
   STATUS[897].EXT.AckRequired := FALSE;
   STATUS[897].EXT.Maintanence := FALSE;
   STATUS[897].EXT.Operation := FALSE;
   STATUS[897].EXT.Forced := FALSE;
   STATUS[897].EXT.BIT29 := FALSE;
   STATUS[897].EXT.BIT30 := FALSE;
   STATUS[897].EXT.BIT31 := FALSE;
   STATUS[897].EXT.ModeBit1 := FALSE;
   STATUS[897].EXT.ModeBit2 := FALSE;
   STATUS[897].EXT.ModeBit3 := FALSE;
   STATUS[897].EXT.BIT19 := FALSE;
   STATUS[897].EXT.BIT20 := FALSE;
   STATUS[897].EXT.AlarmSuppressed := FALSE;
   STATUS[897].EXT.AlarmPrsent := FALSE;
   STATUS[897].EXT.AlarmFailUnAck := FALSE;
   STATUS[897].Status := 0;
   STATUS[897].TimeStamp := 16#0000;
   STATUS[898].VALUE := 0.0;
   STATUS[898].TRIGVALUE := 0.0;
   STATUS[898].EXT.AlarmWarnUnAck := FALSE;
   STATUS[898].EXT.AckRequired := FALSE;
   STATUS[898].EXT.Maintanence := FALSE;
   STATUS[898].EXT.Operation := FALSE;
   STATUS[898].EXT.Forced := FALSE;
   STATUS[898].EXT.BIT29 := FALSE;
   STATUS[898].EXT.BIT30 := FALSE;
   STATUS[898].EXT.BIT31 := FALSE;
   STATUS[898].EXT.ModeBit1 := FALSE;
   STATUS[898].EXT.ModeBit2 := FALSE;
   STATUS[898].EXT.ModeBit3 := FALSE;
   STATUS[898].EXT.BIT19 := FALSE;
   STATUS[898].EXT.BIT20 := FALSE;
   STATUS[898].EXT.AlarmSuppressed := FALSE;
   STATUS[898].EXT.AlarmPrsent := FALSE;
   STATUS[898].EXT.AlarmFailUnAck := FALSE;
   STATUS[898].Status := 0;
   STATUS[898].TimeStamp := 16#0000;
   STATUS[899].VALUE := 0.0;
   STATUS[899].TRIGVALUE := 0.0;
   STATUS[899].EXT.AlarmWarnUnAck := FALSE;
   STATUS[899].EXT.AckRequired := FALSE;
   STATUS[899].EXT.Maintanence := FALSE;
   STATUS[899].EXT.Operation := FALSE;
   STATUS[899].EXT.Forced := FALSE;
   STATUS[899].EXT.BIT29 := FALSE;
   STATUS[899].EXT.BIT30 := FALSE;
   STATUS[899].EXT.BIT31 := FALSE;
   STATUS[899].EXT.ModeBit1 := FALSE;
   STATUS[899].EXT.ModeBit2 := FALSE;
   STATUS[899].EXT.ModeBit3 := FALSE;
   STATUS[899].EXT.BIT19 := FALSE;
   STATUS[899].EXT.BIT20 := FALSE;
   STATUS[899].EXT.AlarmSuppressed := FALSE;
   STATUS[899].EXT.AlarmPrsent := FALSE;
   STATUS[899].EXT.AlarmFailUnAck := FALSE;
   STATUS[899].Status := 0;
   STATUS[899].TimeStamp := 16#0000;
   STATUS[900].VALUE := 0.0;
   STATUS[900].TRIGVALUE := 0.0;
   STATUS[900].EXT.AlarmWarnUnAck := FALSE;
   STATUS[900].EXT.AckRequired := FALSE;
   STATUS[900].EXT.Maintanence := FALSE;
   STATUS[900].EXT.Operation := FALSE;
   STATUS[900].EXT.Forced := FALSE;
   STATUS[900].EXT.BIT29 := FALSE;
   STATUS[900].EXT.BIT30 := FALSE;
   STATUS[900].EXT.BIT31 := FALSE;
   STATUS[900].EXT.ModeBit1 := FALSE;
   STATUS[900].EXT.ModeBit2 := FALSE;
   STATUS[900].EXT.ModeBit3 := FALSE;
   STATUS[900].EXT.BIT19 := FALSE;
   STATUS[900].EXT.BIT20 := FALSE;
   STATUS[900].EXT.AlarmSuppressed := FALSE;
   STATUS[900].EXT.AlarmPrsent := FALSE;
   STATUS[900].EXT.AlarmFailUnAck := FALSE;
   STATUS[900].Status := 0;
   STATUS[900].TimeStamp := 16#0000;
   STATUS[901].VALUE := 0.0;
   STATUS[901].TRIGVALUE := 0.0;
   STATUS[901].EXT.AlarmWarnUnAck := FALSE;
   STATUS[901].EXT.AckRequired := FALSE;
   STATUS[901].EXT.Maintanence := FALSE;
   STATUS[901].EXT.Operation := FALSE;
   STATUS[901].EXT.Forced := FALSE;
   STATUS[901].EXT.BIT29 := FALSE;
   STATUS[901].EXT.BIT30 := FALSE;
   STATUS[901].EXT.BIT31 := FALSE;
   STATUS[901].EXT.ModeBit1 := FALSE;
   STATUS[901].EXT.ModeBit2 := FALSE;
   STATUS[901].EXT.ModeBit3 := FALSE;
   STATUS[901].EXT.BIT19 := FALSE;
   STATUS[901].EXT.BIT20 := FALSE;
   STATUS[901].EXT.AlarmSuppressed := FALSE;
   STATUS[901].EXT.AlarmPrsent := FALSE;
   STATUS[901].EXT.AlarmFailUnAck := FALSE;
   STATUS[901].Status := 0;
   STATUS[901].TimeStamp := 16#0000;
   STATUS[902].VALUE := 0.0;
   STATUS[902].TRIGVALUE := 0.0;
   STATUS[902].EXT.AlarmWarnUnAck := FALSE;
   STATUS[902].EXT.AckRequired := FALSE;
   STATUS[902].EXT.Maintanence := FALSE;
   STATUS[902].EXT.Operation := FALSE;
   STATUS[902].EXT.Forced := FALSE;
   STATUS[902].EXT.BIT29 := FALSE;
   STATUS[902].EXT.BIT30 := FALSE;
   STATUS[902].EXT.BIT31 := FALSE;
   STATUS[902].EXT.ModeBit1 := FALSE;
   STATUS[902].EXT.ModeBit2 := FALSE;
   STATUS[902].EXT.ModeBit3 := FALSE;
   STATUS[902].EXT.BIT19 := FALSE;
   STATUS[902].EXT.BIT20 := FALSE;
   STATUS[902].EXT.AlarmSuppressed := FALSE;
   STATUS[902].EXT.AlarmPrsent := FALSE;
   STATUS[902].EXT.AlarmFailUnAck := FALSE;
   STATUS[902].Status := 0;
   STATUS[902].TimeStamp := 16#0000;
   STATUS[903].VALUE := 0.0;
   STATUS[903].TRIGVALUE := 0.0;
   STATUS[903].EXT.AlarmWarnUnAck := FALSE;
   STATUS[903].EXT.AckRequired := FALSE;
   STATUS[903].EXT.Maintanence := FALSE;
   STATUS[903].EXT.Operation := FALSE;
   STATUS[903].EXT.Forced := FALSE;
   STATUS[903].EXT.BIT29 := FALSE;
   STATUS[903].EXT.BIT30 := FALSE;
   STATUS[903].EXT.BIT31 := FALSE;
   STATUS[903].EXT.ModeBit1 := FALSE;
   STATUS[903].EXT.ModeBit2 := FALSE;
   STATUS[903].EXT.ModeBit3 := FALSE;
   STATUS[903].EXT.BIT19 := FALSE;
   STATUS[903].EXT.BIT20 := FALSE;
   STATUS[903].EXT.AlarmSuppressed := FALSE;
   STATUS[903].EXT.AlarmPrsent := FALSE;
   STATUS[903].EXT.AlarmFailUnAck := FALSE;
   STATUS[903].Status := 0;
   STATUS[903].TimeStamp := 16#0000;
   STATUS[904].VALUE := 0.0;
   STATUS[904].TRIGVALUE := 0.0;
   STATUS[904].EXT.AlarmWarnUnAck := FALSE;
   STATUS[904].EXT.AckRequired := FALSE;
   STATUS[904].EXT.Maintanence := FALSE;
   STATUS[904].EXT.Operation := FALSE;
   STATUS[904].EXT.Forced := FALSE;
   STATUS[904].EXT.BIT29 := FALSE;
   STATUS[904].EXT.BIT30 := FALSE;
   STATUS[904].EXT.BIT31 := FALSE;
   STATUS[904].EXT.ModeBit1 := FALSE;
   STATUS[904].EXT.ModeBit2 := FALSE;
   STATUS[904].EXT.ModeBit3 := FALSE;
   STATUS[904].EXT.BIT19 := FALSE;
   STATUS[904].EXT.BIT20 := FALSE;
   STATUS[904].EXT.AlarmSuppressed := FALSE;
   STATUS[904].EXT.AlarmPrsent := FALSE;
   STATUS[904].EXT.AlarmFailUnAck := FALSE;
   STATUS[904].Status := 0;
   STATUS[904].TimeStamp := 16#0000;
   STATUS[905].VALUE := 0.0;
   STATUS[905].TRIGVALUE := 0.0;
   STATUS[905].EXT.AlarmWarnUnAck := FALSE;
   STATUS[905].EXT.AckRequired := FALSE;
   STATUS[905].EXT.Maintanence := FALSE;
   STATUS[905].EXT.Operation := FALSE;
   STATUS[905].EXT.Forced := FALSE;
   STATUS[905].EXT.BIT29 := FALSE;
   STATUS[905].EXT.BIT30 := FALSE;
   STATUS[905].EXT.BIT31 := FALSE;
   STATUS[905].EXT.ModeBit1 := FALSE;
   STATUS[905].EXT.ModeBit2 := FALSE;
   STATUS[905].EXT.ModeBit3 := FALSE;
   STATUS[905].EXT.BIT19 := FALSE;
   STATUS[905].EXT.BIT20 := FALSE;
   STATUS[905].EXT.AlarmSuppressed := FALSE;
   STATUS[905].EXT.AlarmPrsent := FALSE;
   STATUS[905].EXT.AlarmFailUnAck := FALSE;
   STATUS[905].Status := 0;
   STATUS[905].TimeStamp := 16#0000;
   STATUS[906].VALUE := 0.0;
   STATUS[906].TRIGVALUE := 0.0;
   STATUS[906].EXT.AlarmWarnUnAck := FALSE;
   STATUS[906].EXT.AckRequired := FALSE;
   STATUS[906].EXT.Maintanence := FALSE;
   STATUS[906].EXT.Operation := FALSE;
   STATUS[906].EXT.Forced := FALSE;
   STATUS[906].EXT.BIT29 := FALSE;
   STATUS[906].EXT.BIT30 := FALSE;
   STATUS[906].EXT.BIT31 := FALSE;
   STATUS[906].EXT.ModeBit1 := FALSE;
   STATUS[906].EXT.ModeBit2 := FALSE;
   STATUS[906].EXT.ModeBit3 := FALSE;
   STATUS[906].EXT.BIT19 := FALSE;
   STATUS[906].EXT.BIT20 := FALSE;
   STATUS[906].EXT.AlarmSuppressed := FALSE;
   STATUS[906].EXT.AlarmPrsent := FALSE;
   STATUS[906].EXT.AlarmFailUnAck := FALSE;
   STATUS[906].Status := 0;
   STATUS[906].TimeStamp := 16#0000;
   STATUS[907].VALUE := 0.0;
   STATUS[907].TRIGVALUE := 0.0;
   STATUS[907].EXT.AlarmWarnUnAck := FALSE;
   STATUS[907].EXT.AckRequired := FALSE;
   STATUS[907].EXT.Maintanence := FALSE;
   STATUS[907].EXT.Operation := FALSE;
   STATUS[907].EXT.Forced := FALSE;
   STATUS[907].EXT.BIT29 := FALSE;
   STATUS[907].EXT.BIT30 := FALSE;
   STATUS[907].EXT.BIT31 := FALSE;
   STATUS[907].EXT.ModeBit1 := FALSE;
   STATUS[907].EXT.ModeBit2 := FALSE;
   STATUS[907].EXT.ModeBit3 := FALSE;
   STATUS[907].EXT.BIT19 := FALSE;
   STATUS[907].EXT.BIT20 := FALSE;
   STATUS[907].EXT.AlarmSuppressed := FALSE;
   STATUS[907].EXT.AlarmPrsent := FALSE;
   STATUS[907].EXT.AlarmFailUnAck := FALSE;
   STATUS[907].Status := 0;
   STATUS[907].TimeStamp := 16#0000;
   STATUS[908].VALUE := 0.0;
   STATUS[908].TRIGVALUE := 0.0;
   STATUS[908].EXT.AlarmWarnUnAck := FALSE;
   STATUS[908].EXT.AckRequired := FALSE;
   STATUS[908].EXT.Maintanence := FALSE;
   STATUS[908].EXT.Operation := FALSE;
   STATUS[908].EXT.Forced := FALSE;
   STATUS[908].EXT.BIT29 := FALSE;
   STATUS[908].EXT.BIT30 := FALSE;
   STATUS[908].EXT.BIT31 := FALSE;
